ABB RAPID module: Rob2_MainModule.mod

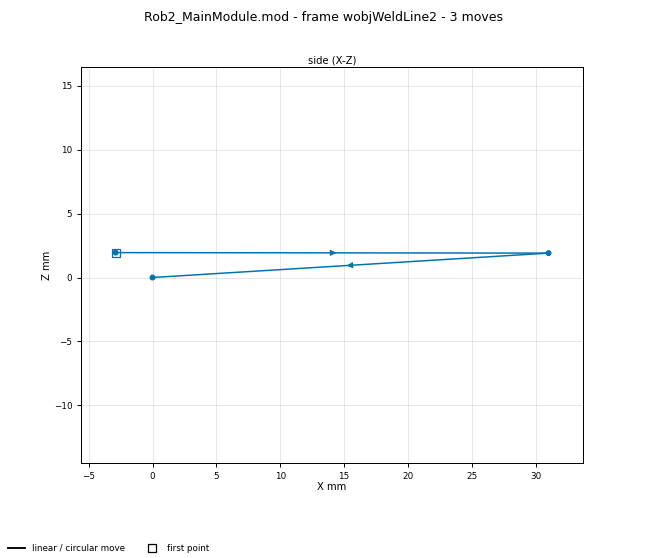
[picture p0: tool path of Rob2_MainModule.mod in frame wobjWeldLine2, 3 of 41 moves have a stored position in this frame; points joined in program order, loops and branches not executed]
MODULE Rob2_MainModule
	!========================================
	! TASK2 (Robot2) - Rob2_MainModule
	! Version History
	!========================================
	! v1.9.44 (2026-02-24) - FIX: Restore MoveAbsJ in MoveJgJ for home return
	!   - ROOT CAUSE: v1.9.42 removed robot motion from MoveJgJ
	!     T_Head rMoveToRobotHome sends robot joint targets via jRob2 PERS
	!     but Robot2 ignored them, causing home return to not move robots
	!   - FIX: MoveAbsJ jRob2, vSync, fine, tool0 restored
	!     MoveAbsJ is joint-space; tool0 vs tWeld2 does not affect joint angles
	!     MergeJgWith() defaults to CJointT for unspecified axes (backward compatible)
	!
	! v1.9.43 (2026-02-21) - Floor coordinate TCP logging
	!   - Added CRobT(\Tool:=tWeld2\WObj:=WobjFloor) to SetRobot2InitialPosition
	!   - Logs TCP_Floor position + orientation to robot2_init_position.txt
	!   - For verifying Robot1/Robot2 TCP meeting point at R-axis center
	!
	! v1.9.42 (2026-02-19) - MoveJgJ fix for tWeld2 [REVERTED in v1.9.44]
	!   - Removed MoveAbsJ jRob2 from MoveJgJ case
	!   - jRob2.robax is tool0-calculated (138deg J2 change from tWeld2 HOME)
	!   - Robot2 now immediately Acks without moving during gantry move
	!   - Prevents concurrent MoveAbsJ conflict with Robot1
	!
	! v2.1.0 (2026-02-03)
	!   - Added PlanA-style command monitoring loop
	!   - Robot2_CommandLoop() monitors nCmdInput from ConfigModule
	!   - TEST_MODE=10 enters real-time command monitoring
	!   - Responds to CMD_WELD, CMD_EDGE_WELD, CMD_ROB2_WIRE_CUT
	!
	! v1.0.0 (2025-12-17)
	!   - Initial gantry position sharing system
	!   - Added shared_gantry_pos and related variables
	!   - Created UpdateSharedGantryPosition procedure
	!
	! v1.1.0 (2025-12-18)
	!   - Added wobj0 definition verification
	!   - Verified Robot2's wobj0 is READ-ONLY (equals World)
	!   - Documented wobj0 vs WobjFloor relationship
	!
	! v1.2.0 (2025-12-18)
	!   - Added WobjFloor coordinate system
	!   - Frame: [-9500, 5300, 2100] with quaternion [0, 1, 0, 0]
	!   - Quaternion [0,1,0,0] = 180deg rotation around X-axis (Y,Z inverted)
	!   - Added comprehensive coordinate system documentation
	!
	! v1.3.0 (2025-12-18)
	!   - Added coordinate verification procedures
	!   - TestRobot2_TCP: TCP position verification in wobj0 and WobjFloor
	!   - TestRobot2_XYZ: X/Y/Z axis movement tests
	!   - TestCoordinateMovement: Core movement and logging procedure
	!   - WritePosToFile: File logging with overwrite mode
	!
	! v1.4.0 (2025-12-18)
	!   - Added World coordinate comparison
	!   - CompareRobot2Coordinates: Compare wobj0, WobjFloor, World
	!   - Verified relationship: wobj0 = World (for Robot2)
	!   - Verified WobjFloor transforms coordinates correctly
	!
	! v1.4.1 (2025-12-23)
	!   - Removed MoveToMiddlePosition calls to prevent Reference Error
	!   - Simplified procedure calls in TestRobot2_TCP
	!
	! v1.4.2 (2025-12-24)
	!   - Added Robot2 TCP coordinate movement tests
	!   - TestCoordinateMovement: Move and log TCP positions
	!
	! v1.4.3 (2025-12-24)
	!   - Combined X/Y/Z tests into single TestRobot2_XYZ procedure
	!   - Streamlined coordinate testing workflow
	!
	! v1.4.4 (2025-12-24)
	!   - Reduced movement distance to avoid joint limits
	!   - Changed test distances: 50mm X, 30mm Y, 20mm Z
	!
	! v1.4.5 (2025-12-24)
	!   - Increased movement back to 50/30/20 mm
	!   - Added return to start position after test
	!
	! v1.4.6 (2025-12-24)
	!   - Added home position test capability
	!   - Save original joint position with CJointT()
	!   - Move to home position [0,0,0,0,0,0] before test
	!   - Return to original position after test
	!
	! v1.4.7 (2025-12-24)
	!   - Fixed singularity error in home position
	!   - Changed Robot2 home position to [+90,0,0,0,30,0]
	!   - J1=+90deg for Robot2 mounting orientation
	!   - J5=30deg to avoid wrist singularity (not 0deg)
	!
	! v1.5.0 (2025-12-24) - DUAL COORDINATE SYSTEM
	!   - Added config.txt MODE support for dual coordinate systems
	!   - ReadConfigMode() function reads /HOME/config.txt
	!   - MODE=0 (Default - User's system):
	!     * Robot2 uses WobjFloor as base coordinate
	!     * wobj0 [+50,+30,+20] -> Floor [+50,+30,+20] (NO Y,Z inversion)
	!   - MODE=1 (Claude's system):
	!     * Robot2 uses wobj0 as base coordinate
	!     * wobj0 [+50,+30,+20] -> Floor [+50,-30,-20] (Y,Z inverted)
	!   - Modified TestCoordinateMovement to accept wobjdata parameter
	!   - TestRobot2_XYZ now switches coordinate system based on MODE
	!
	! v1.7.45 - v1.7.47 (2025-12-31)
	!   - Updated SetRobot2InitialPosition to match Robot1 HOME position
	!   - Robot2 HOME: TCP [0, 488, -1000] with quaternion [0.50000, -0.50000, -0.50000, -0.50000]
	!   - Fixed 40512 error using actual extax values from CJointT()
	!
	! v1.7.50 (2025-12-31)
	!   - Added WobjGantry_Rob2 dynamic work object for Robot2 TCP control
	!   - Implemented UpdateGantryWobj_Rob2() to read gantry position from TASK1
	!   - Robot2 cannot control gantry - must use CJointT(\TaskName:="T_ROB1")
	!   - R-axis rotation with 90deg base offset (R=0: gantry parallel to Y-axis)
	!   - Enables Robot2 TCP control in Floor coordinates regardless of gantry position
	!   - SetRobot2InitialPosition now uses WobjGantry_Rob2 instead of wobj0
	!========================================

    RECORD targetdata
        robtarget position;
        num cpm;
        num schedule;
        num voltage;
        num wfs;
        num Current;
        num WeaveShape;
        num WeaveType;
        num WeaveLength;
        num WeaveWidth;
        num WeaveDwellLeft;
        num WeaveDwellRight;
        num TrackType;
        num TrackGainY;
        num TrackGainZ;
        num MaxCorr;
        num Bias;
    ENDRECORD

    RECORD monRobs
        extjoint monExt;
        robjoint monJoint1;
        robjoint monJoint2;
        pose monPose1;
        pose monPose2;
    ENDRECORD

    RECORD torchmotion
        num No;
        num LengthOffset;
        num BreadthOffset;
        num HeightOffset;
        num WorkingAngle;
        num TravelAngle;
        num WeldingSpeed;
        num Schedule;
        num Voltage;
        num FeedingSpeed;
        num Current;
        num WeaveShape;
        num WeaveType;
        num WeaveLength;
        num WeaveWidth;
        num WeaveDwellLeft;
        num WeaveDwellRight;
        num TrackType;
        num TrackGainY;
        num TrackGainZ;
        num MaxCorr;
        num Bias;
    ENDRECORD

    RECORD corrorder
        num X_StartOffset;
        num X_Depth;
        num X_ReturnLength;
        num Y_StartOffset;
        num Y_Depth;
        num Y_ReturnLength;
        num Z_StartOffset;
        num Z_Depth;
        num Z_ReturnLength;
        num RY_Torch;
    ENDRECORD

    RECORD edgedata
        pos EdgePos;
        num Height;
        num Breadth;
        num HoleSize;
        num Thickness;
        num AngleHeight;
        num AngleWidth;
    ENDRECORD

	! v1.7.51 (2026-01-03)
	!   - Added robot2_init_complete synchronization flag
	!   - TASK2 sets flag to TRUE after SetRobot2InitialPosition completes
	!   - Enables precise TASK1/TASK2 synchronization without fixed delays
	!   - Replaces crude WaitTime 10.0 approach with event-based signaling
	!
	! v1.8.0 (2026-01-03)
	!   - Version sync with TASK1 for R-axis rotation testing
	!   - No functional changes in TASK2 (changes in TASK1 only)
	!   - Ready for Phase 2: Complex motion testing
	!
	! v1.8.7 (2026-01-05)
	!   - FIX: Use gantry extax from TASK1 for Robot2 MoveJ/MoveL in SetRobot2InitialPosition.
	!
	! v1.8.9 (2026-01-05)
	!   - STABILITY: Reduced TPWrite output and file writes in SetRobot2InitialPosition.
	!
	! v1.8.10 (2026-01-05)
	!   - FEAT: Added TEST_MODE=2 Robot2 TCP offset move from config.txt.
	!
	! v1.8.11 (2026-01-06)
	!   - FIX: Guard config parsing in SetRobot2OffsetPosition to avoid StrPart errors.
	!
	! v1.8.12 (2026-01-06)
	!   - FIX: Allow missing TCP_OFFSET_* with default 0 values.
	!
	! v1.8.13 (2026-01-06)
	!   - Version sync with TASK1 (Mode2 range checks).
	!
	! v1.8.14 (2026-01-06)
	!   - Version sync with TASK1 (MOC.cfg range update).
	!
	! v1.8.15 (2026-01-06)
	!   - FIX: Use TASK PERS for robot1_floor_pos_t2 to avoid global PERS ambiguity.
	!
	! v1.8.16 (2026-01-06)
	!   - FIX: Initialize TASK PERS robot1_floor_pos_t2 to satisfy RAPID syntax.
	!
	! v1.8.18 (2026-01-06)
	!   - Version sync with TASK1 (robot1_floor_pos_t1 rename in TASK1).
	!
	! v1.8.19 (2026-01-06)
	!   - Version sync with TASK1 (robot2_floor_pos_t1 rename in TASK1).
	!
	! v1.8.20 (2026-01-06)
	!   - FIX: Rename robot2_floor_pos to robot2_floor_pos_t1 and remove initializer.
	!
	! v1.8.21 (2026-01-06)
	!   - Version sync with TASK1 (Mode2 gantry HOME return).
	!
	! v1.8.22 (2026-01-06)
	!   - FEAT: Support per-robot TCP offsets (R2) for Mode2 via TCP_OFFSET_R2_*.
	!
	! v1.8.23 (2026-01-07)
	!   - FIX: Make Mode2 TCP offset parsing tolerant of leading whitespace.
	!
	! v1.8.24 (2026-01-07)
	!   - Version sync with TASK1 (Mode2 TCP offset debug logging).
	!
	! v1.8.25 (2026-01-07)
	!   - Version sync with TASK1 (ignore comment lines during offset parse).
	!
	! v1.8.26 (2026-01-07)
	!   - Version sync with TASK1 (trim leading whitespace during offset parse).
	!
	! v1.8.27 (2026-01-07)
	!   - Version sync with TASK1 (remove tab escape in trim loop).
	!
	! v1.8.28 (2026-01-07)
	!   - Version sync with TASK1 (remove RemoveCR in offset parse loop).
	!
	! v1.8.29 (2026-01-07)
	!   - Version sync with TASK1 (remove RemoveCR in offset parse loop).
	!
! v1.8.31 (2026-01-07)
!   - FIX: Use TASK PERS for robot2_init_complete to share flag with TASK1.
!   - FIX: Set robot2_init_complete right after Step1 to avoid TASK1 timeout.
!   - FIX: Add EOF-safe config parsing in ReadTestMode and Mode2 offset parse.
!   - DIAG: Log Mode2 offset start in main process.
!
! v1.8.32 (2026-01-08)
!   - Version sync with TASK1 (robot2_init_complete init in TASK1).
!
! v1.8.33 (2026-01-08)
!   - DIAG: Log entry at start of TASK2 main before config read.
!
! v1.8.34 (2026-01-08)
!   - DIAG: Bypass ReadTestMode temporarily (force TEST_MODE=2).
!
! v1.8.35 (2026-01-08)
!   - FIX: Revert robot2_init_complete to shared PERS for cross-task sync.
!
! v1.8.36 (2026-01-08)
!   - DIAG: Log Mode2 offset inputs, gantry extax, and target TCP before MoveJ.
!
! v1.8.37 (2026-01-08)
!   - DIAG: Create Mode2 offset log at entry before config parsing.
!
! v1.8.38 (2026-01-08)
!   - FIX: Guard comment detection to avoid StrPart on empty strings in config parse.
!
! v1.8.39 (2026-01-08)
!   - FIX - Read Mode2 TCP offsets from TASK1 shared PERS (no config read).
!
! v1.8.55 (2026-01-12)
!   - FIX - Remove 488mm from offset_tcp calculation
!   - CAUSE - MoveJ uses WobjGantry_Rob2 (R-center reference)
!   - 488mm was only needed for wobj0 reference, not WobjGantry_Rob2
!   - RESULT - TCP distance 200mm fixed (R-angle independent)
	!
	! v1.8.30 (2026-01-07)
	!   - Version sync with TASK1 (stop offset parse once keys are found).
	!
	! v1.8.17 (2026-01-06)
	!   - FIX: Rename TASK2 local copy to robot1_floor_pos_t2 to avoid PERS ambiguity.
	!
	! v1.8.8 (2026-01-05)
	!   - STABILITY: Reduced main process log writes to lower 41617 risk.
	!
	! v1.8.5 (2026-01-04)
	!   - Version synchronized with TASK1 (Robot2 angle correction in TASK1).
	!   - No functional changes in TASK2.
	!
	! v1.8.3 (2026-01-04)
	!   - STABILITY: Added ERROR handlers to main and SetRobot2InitialPosition
	!   - STABILITY: Corrected file handle usage in 4 procedures (single Open statement)
	!   - STANDARDS: Replaced Unicode characters (deg symbol) with ASCII equivalents
	!   - STANDARDS: Changed file encoding from UTF-8 to ASCII
	!   - Version synchronized with TASK1 (jumped from v1.8.0)
	!
! Version constant for logging (v1.8.39+)
CONST string TASK2_VERSION := "v1.9.46";

! Synchronization flag for TASK1/TASK2 initialization
! TASK2 sets this to TRUE when Robot2 initialization is complete
! TASK1 waits for this flag before starting gantry floor tests
PERS bool robot2_init_complete;
! Mode2 TCP offsets for Robot2 (shared from TASK1)
PERS num mode2_r2_offset_x;
PERS num mode2_r2_offset_y;
PERS num mode2_r2_offset_z;

! v1.8.57: Synchronization flag - wait for TASK1 to update config values
PERS bool mode2_config_ready;

! v1.8.63: Robot2 reposition sync flags
PERS bool mode2_r2_reposition_trigger;
PERS bool mode2_r2_reposition_done;
! v1.8.67: Initial offset complete flag
PERS bool mode2_r2_initial_offset_done;

! v1.9.17: Shared test_mode from TASK1
PERS num shared_test_mode;

! v2.1.0: Command Interface Variables (shared with TASK1 ConfigModule)
PERS num nCmdInput;
PERS num nCmdOutput;
PERS num nCmdMatch;

! v2.1.0: Command Constants (must match TASK1 ConfigModule)
CONST num CMD_MOVE_TO_WORLDHOME := 101;
CONST num CMD_WELD := 200;
CONST num CMD_WELD_MOTION := 201;
CONST num CMD_EDGE_WELD := 210;
CONST num CMD_ROB2_WIRE_CUT := 512;

! v1.8.70: Store Robot2 offset joints (like robot1_offset_joints in TASK1)
! Initial call: MoveJ then save joints
! Reposition call: Skip MoveJ (joints already at offset, gantry moved)
VAR robjoint robot2_offset_joints;

    PERS tasks taskGroup12{2};
    PERS tasks taskGroup13{2};
    PERS tasks taskGroup23{2};
    PERS tasks taskGroup123{3};
    PERS pos nCaledR2Pos;
    TASK PERS jointtarget jTemp:=[[0,-2.51761,-12.1411,0,15.6587,0],[-500,500,300,15,0,-28.6479]];
    PERS wobjdata wobjtest:=[FALSE,TRUE,"GantryRob",[[-971.372,373.696,300],[1,0,0,0]],[[0,0,0],[1,0,0,0]]];

    ! Sync Data
    TASK VAR syncident SynchronizeJGJon{9999};
    TASK VAR syncident SynchronizePGJon{9999};
    TASK VAR syncident SynchronizePGLon{9999};
    TASK VAR syncident SynchronizeJGJoff{9999};
    TASK VAR syncident SynchronizePGJoff{9999};
    TASK VAR syncident SynchronizePGLoff{9999};
    TASK VAR syncident Wait{100};

    PERS string stCommand;
    PERS string stReact{3};
    PERS num idSync;
    PERS speeddata vSync;
    PERS zonedata zSync;

    PERS wobjdata wobjWeldLine2;
    PERS wobjdata wobjRotCtr2;

    ! Weld Sequence Sync Variables (v1.9.0)
    ! Cross-task synchronization with TASK1
    PERS bool t2_weld_ready;    ! Robot2 ready signal (set by TASK2)
    PERS bool t1_weld_start;    ! TASK1 weld start signal (read by TASK2)
    PERS bool t1_weld_done;     ! TASK1 weld done signal (read by TASK2)

    ! Edge-based Weld Sequence Sync Variables (v2.0.0)
    ! From TASK1 MainModule
    PERS bool t1_weld_position_ready;  ! TASK1 gantry+Robot1 positioned
    PERS bool shared_bRobSwap;         ! Robot swap flag from TASK1

    ! Robot2 edge positions (shared from TASK1, v1.9.37)
    PERS pos shared_posStart_r2;
    PERS pos shared_posEnd_r2;
    PERS num shared_nLengthWeldLine;

    ! stCommand/stReact Protocol (v1.9.39 - T_Head interface)
    ! T_Head sets stCommand, TASK1/2 respond via stReact
    ! NOTE: stCommand/stReact already declared above (lines 361-362)

    ! Weld WObj for Robot2 (v1.9.0)
    ! Created by TASK1, referenced by TASK2
    PERS wobjdata WobjWeldR2;

    ! Robot2 Weld Orientation from ConfigModule (v1.9.0)
    ! Cross-task reference to TASK1 ConfigModule
    PERS num WELD_R2_ORIENT_Q1;
    PERS num WELD_R2_ORIENT_Q2;
    PERS num WELD_R2_ORIENT_Q3;
    PERS num WELD_R2_ORIENT_Q4;

    ! Robot2 Weld Position in WObj (v1.9.1)
    ! Cross-task reference to TASK1 ConfigModule
    ! WObj: X=weld direction, Y=perpendicular, Z=Floor Z
    PERS num WELD_R2_WObj_X;
    PERS num WELD_R2_WObj_Y;
    PERS num WELD_R2_WObj_Z;

    ! Work Object Definitions (v1.7.13 2025-12-28)
    ! WobjFloor: Floor coordinate system from TASK1 (external reference)
    PERS wobjdata WobjFloor;

    ! WobjFloor_Rob2: Floor coordinate system for Robot2
    ! MUST be identical to TASK1's WobjFloor (absolute world coordinate)
    ! uframe: [-9500, 5300, 2100] = Gantry HOME in Floor coordinate
    ! rot: [1, 0, 0, 0] = No rotation (Robot2 wobj0 aligned with Floor!)
    PERS wobjdata WobjFloor_Rob2 := [FALSE, TRUE, "", [[-9500, 5300, 2100], [1, 0, 0, 0]], [[0, 0, 0], [1, 0, 0, 0]]];

    ! WobjGantry_Rob2: Dynamic work object for Robot2 TCP control (v1.7.50)
    ! Updated by UpdateGantryWobj_Rob2() to track gantry position from TASK1
    ! Allows Robot2 TCP control in Floor coordinates regardless of gantry position
    ! Robot2 cannot control gantry, must read position from TASK1
    PERS wobjdata WobjGantry_Rob2 := [FALSE, TRUE, "", [[0, 0, 0], [1, 0, 0, 0]], [[0, 0, 0], [1, 0, 0, 0]]];

    ! WobjRobot2Base_Dynamic: Robot2 base coordinate from TASK1 (external reference) (v1.7.50)
    ! TASK1 updates this to track Robot2 base position as gantry moves
    ! Robot2 uses this to calculate its Floor TCP position
    ! Direction = Floor direction (no rotation, quaternion [1,0,0,0])
    PERS wobjdata WobjRobot2Base_Dynamic;

    ! wobjRob2Base: Robot2 Base Frame orientation from MOC.cfg
    ! Quaternion [-4.32964E-17, 0.707107, 0.707107, 4.32964E-17] = 45deg rotation
    PERS wobjdata wobjRob2Base := [FALSE, TRUE, "", [[0, 0, 0], [-0.0000000000000000432964, 0.707107, 0.707107, 0.0000000000000000432964]], [[0, 0, 0], [1, 0, 0, 0]]];

    ! Robot Position Monitoring (v1.5.1 2025-12-25)
    ! Robot1 TCP position from TASK1 (local copy for TASK2)
    TASK PERS robtarget robot1_floor_pos_t2 := [[0,0,0],[1,0,0,0],[0,0,0,0],[0,0,0,0,0,0]];
    ! Robot1 wobj0 snapshot from TASK1 (external reference)
    PERS wobjdata robot1_wobj0_snapshot := [FALSE, TRUE, "", [[0,0,0],[1,0,0,0]], [[0,0,0],[1,0,0,0]]];

    ! Robot2 TCP position in Floor coordinate system (for distance measurement)
    ! Shared across tasks - use PERS (not TASK PERS) for cross-task access
    PERS robtarget robot2_floor_pos_t1;

    PERS num nMotionTotalStep{2};
    PERS num nMotionStepCount{2};
    PERS num nMotionStartStepLast{2};
    PERS num nMotionEndStepLast{2};
    PERS num nRunningStep{2};
    PERS num nWeldSequence;

    PERS jointtarget jRob2;
    PERS robtarget pRob2;
    PERS bool bRqMoveG_PosHold;

    PERS robtarget pctWeldPosR1;
    PERS robtarget pctWeldPosR2;

    PERS targetdata Welds2{40};
    TASK PERS speeddata vWeld{40}:=[[10,200,200,200],[10,200,200,200],[10,200,200,200],[10,200,200,200],[9.16667,200,200,200],[9.16667,200,200,200],[8.33333,200,200,200],[7.5,200,200,200],[0,0,0,0],[0,0,0,0],[0,0,0,0],[0,0,0,0],[0,0,0,0],[0,0,0,0],[0,0,0,0],[0,0,0,0],[0,0,0,0],[0,0,0,0],[0,0,0,0],[0,0,0,0],[0,0,0,0],[0,0,0,0],[0,0,0,0],[0,0,0,0],[0,0,0,0],[0,0,0,0],[0,0,0,0],[0,0,0,0],[0,0,0,0],[0,0,0,0],[0,0,0,0],[0,0,0,0],[0,0,0,0],[0,0,0,0],[0,0,0,0],[0,0,0,0],[0,0,0,0],[0,0,0,0],[0,0,0,0],[10,200,200,200]];
    PERS seamdata smDefault_2{2};


    PERS speeddata vTargetSpeed;
    PERS zonedata zTargetZone;

    TASK PERS welddata wdTrap:=[10,0,[5,0,38,240,0,400,0,0,0],[0,0,0,0,0,0,0,0,0]];
    TASK PERS welddata wd1:=[10,0,[5,0,39.5,260,0,0,0,0,0],[0,0,0,0,0,0,0,0,0]];
    TASK PERS welddata wd2:=[10,0,[5,0,39.5,260,0,0,0,0,0],[0,0,0,0,0,0,0,0,0]];
    TASK PERS welddata wd3:=[10,0,[5,0,39.5,260,0,0,0,0,0],[0,0,0,0,0,0,0,0,0]];
    TASK PERS welddata wd4:=[10,0,[5,0,39.5,260,0,0,0,0,0],[0,0,0,0,0,0,0,0,0]];
    TASK PERS welddata wd5:=[9.16667,0,[5,0,39.5,255,0,420,0,0,0],[0,0,0,0,0,0,0,0,0]];
    TASK PERS welddata wd6:=[9.16667,0,[5,0,39.5,255,0,420,0,0,0],[0,0,0,0,0,0,0,0,0]];
    TASK PERS welddata wd7:=[8.33333,0,[5,0,39.5,255,0,420,0,0,0],[0,0,0,0,0,0,0,0,0]];
    TASK PERS welddata wd8:=[7.5,0,[5,0,36,225,0,375,0,0,0],[0,0,0,0,0,0,0,0,0]];
    TASK PERS welddata wd9:=[7.5,0,[5,0,36,225,0,375,0,0,0],[0,0,0,0,0,0,0,0,0]];
    TASK PERS welddata wd10:=[0,0,[5,0,0,0,0,0,0,0,0],[0,0,0,0,0,0,0,0,0]];
    TASK PERS welddata wd11:=[0,0,[5,0,0,0,0,0,0,0,0],[0,0,0,0,0,0,0,0,0]];
    TASK PERS welddata wd12:=[0,0,[5,0,0,0,0,0,0,0,0],[0,0,0,0,0,0,0,0,0]];
    TASK PERS welddata wd13:=[0,0,[5,0,0,0,0,0,0,0,0],[0,0,0,0,0,0,0,0,0]];
    TASK PERS welddata wd14:=[0,0,[5,0,0,0,0,0,0,0,0],[0,0,0,0,0,0,0,0,0]];
    TASK PERS welddata wd15:=[0,0,[5,0,0,0,0,0,0,0,0],[0,0,0,0,0,0,0,0,0]];
    TASK PERS welddata wd16:=[0,0,[5,0,0,0,0,0,0,0,0],[0,0,0,0,0,0,0,0,0]];
    TASK PERS welddata wd17:=[0,0,[5,0,0,0,0,0,0,0,0],[0,0,0,0,0,0,0,0,0]];
    TASK PERS welddata wd18:=[0,0,[5,0,0,0,0,0,0,0,0],[0,0,0,0,0,0,0,0,0]];
    TASK PERS welddata wd19:=[0,0,[5,0,0,0,0,0,0,0,0],[0,0,0,0,0,0,0,0,0]];
    TASK PERS welddata wd20:=[0,0,[5,0,0,0,0,0,0,0,0],[0,0,0,0,0,0,0,0,0]];
    TASK PERS welddata wd21:=[0,0,[5,0,0,0,0,0,0,0,0],[0,0,0,0,0,0,0,0,0]];
    TASK PERS welddata wd22:=[0,0,[5,0,0,0,0,0,0,0,0],[0,0,0,0,0,0,0,0,0]];
    TASK PERS welddata wd23:=[0,0,[5,0,0,0,0,0,0,0,0],[0,0,0,0,0,0,0,0,0]];
    TASK PERS welddata wd24:=[0,0,[5,0,0,0,0,0,0,0,0],[0,0,0,0,0,0,0,0,0]];
    TASK PERS welddata wd25:=[0,0,[5,0,0,0,0,0,0,0,0],[0,0,0,0,0,0,0,0,0]];
    TASK PERS welddata wd26:=[0,0,[5,0,0,0,0,0,0,0,0],[0,0,0,0,0,0,0,0,0]];
    TASK PERS welddata wd27:=[0,0,[5,0,0,0,0,0,0,0,0],[0,0,0,0,0,0,0,0,0]];
    TASK PERS welddata wd28:=[0,0,[5,0,0,0,0,0,0,0,0],[0,0,0,0,0,0,0,0,0]];
    TASK PERS welddata wd29:=[0,0,[5,0,0,0,0,0,0,0,0],[0,0,0,0,0,0,0,0,0]];
    TASK PERS welddata wd30:=[0,0,[5,0,0,0,0,0,0,0,0],[0,0,0,0,0,0,0,0,0]];
    TASK PERS welddata wd31:=[0,0,[5,0,0,0,0,0,0,0,0],[0,0,0,0,0,0,0,0,0]];
    TASK PERS welddata wd32:=[0,0,[5,0,0,0,0,0,0,0,0],[0,0,0,0,0,0,0,0,0]];
    TASK PERS welddata wd33:=[0,0,[5,0,0,0,0,0,0,0,0],[0,0,0,0,0,0,0,0,0]];
    TASK PERS welddata wd34:=[0,0,[5,0,0,0,0,0,0,0,0],[0,0,0,0,0,0,0,0,0]];
    TASK PERS welddata wd35:=[0,0,[5,0,0,0,0,0,0,0,0],[0,0,0,0,0,0,0,0,0]];
    TASK PERS welddata wd36:=[0,0,[5,0,0,0,0,0,0,0,0],[0,0,0,0,0,0,0,0,0]];
    TASK PERS welddata wd37:=[0,0,[5,0,0,0,0,0,0,0,0],[0,0,0,0,0,0,0,0,0]];
    TASK PERS welddata wd38:=[0,0,[5,0,0,0,0,0,0,0,0],[0,0,0,0,0,0,0,0,0]];
    TASK PERS welddata wd39:=[0,0,[5,0,0,0,0,0,0,0,0],[0,0,0,0,0,0,0,0,0]];
    TASK PERS welddata wd40:=[10,0,[5,0,39.5,260,0,0,0,0,0],[0,0,0,0,0,0,0,0,0]];

    TASK PERS welddata Holdwd1:=[0.01,0,[5,0,39.5,260,0,0,0,0,0],[0,0,0,0,0,0,0,0,0]];
    TASK PERS welddata Holdwd2:=[0.01,0,[5,0,39.5,260,0,0,0,0,0],[0,0,0,0,0,0,0,0,0]];
    TASK PERS welddata Holdwd3:=[0.01,0,[5,0,39.5,260,0,0,0,0,0],[0,0,0,0,0,0,0,0,0]];
    TASK PERS welddata Holdwd4:=[0.01,0,[5,0,39.5,260,0,0,0,0,0],[0,0,0,0,0,0,0,0,0]];
    TASK PERS welddata Holdwd5:=[0.01,0,[5,0,39.5,255,0,420,0,0,0],[0,0,0,0,0,0,0,0,0]];
    TASK PERS welddata Holdwd6:=[0.01,0,[5,0,39.5,255,0,420,0,0,0],[0,0,0,0,0,0,0,0,0]];
    TASK PERS welddata Holdwd7:=[0.01,0,[5,0,39.5,255,0,420,0,0,0],[0,0,0,0,0,0,0,0,0]];
    TASK PERS welddata Holdwd8:=[0.01,0,[5,0,36,225,0,375,0,0,0],[0,0,0,0,0,0,0,0,0]];
    TASK PERS welddata Holdwd9:=[0.01,0,[5,0,36,225,0,375,0,0,0],[0,0,0,0,0,0,0,0,0]];
    TASK PERS welddata Holdwd10:=[0.01,0,[5,0,0,0,0,0,0,0,0],[0,0,0,0,0,0,0,0,0]];

    !!! weave data !!!
    TASK PERS weavedata weaveTrap:=[1,2,3,3,0,0,0,0,0,0,0,0,0,0,0];
    TASK PERS weavedata weave1:=[1,2,2,3,0,0,0,0,0,0,0,0,0,0,0];
    TASK PERS weavedata weave2:=[1,2,2,3,0,0,0,0,0,0,0,0,0,0,0];
    TASK PERS weavedata weave3:=[1,2,2,3,0,0,0,0,0,0,0,0,0,0,0];
    TASK PERS weavedata weave4:=[1,2,2,3,0,0,0,0,0,0,0,0,0,0,0];
    TASK PERS weavedata weave5:=[1,2,2,3.5,0,0,0,0,0,0,0,0,0,0,0];
    TASK PERS weavedata weave6:=[1,2,2,3.5,0,0,0,0,0,0,0,0,0,0,0];
    TASK PERS weavedata weave7:=[1,2,2,3.5,0,0,0,0,0,0,0,0,0,0,0];
    TASK PERS weavedata weave8:=[1,0,0,0,0,0,0,0,0,0,0,0,0,0,0];
    TASK PERS weavedata weave9:=[1,0,0,0,0,0,0,0,0,0,0,0,0,0,0];
    TASK PERS weavedata weave10:=[0,0,0,0,0,0,0,0,0,0,0,0,0,0,0];
    TASK PERS weavedata weave11:=[0,0,0,0,0,0,0,0,0,0,0,0,0,0,0];
    TASK PERS weavedata weave12:=[0,0,0,0,0,0,0,0,0,0,0,0,0,0,0];
    TASK PERS weavedata weave13:=[0,0,0,0,0,0,0,0,0,0,0,0,0,0,0];
    TASK PERS weavedata weave14:=[0,0,0,0,0,0,0,0,0,0,0,0,0,0,0];
    TASK PERS weavedata weave15:=[0,0,0,0,0,0,0,0,0,0,0,0,0,0,0];
    TASK PERS weavedata weave16:=[0,0,0,0,0,0,0,0,0,0,0,0,0,0,0];
    TASK PERS weavedata weave17:=[0,0,0,0,0,0,0,0,0,0,0,0,0,0,0];
    TASK PERS weavedata weave18:=[0,0,0,0,0,0,0,0,0,0,0,0,0,0,0];
    TASK PERS weavedata weave19:=[0,0,0,0,0,0,0,0,0,0,0,0,0,0,0];
    TASK PERS weavedata weave20:=[0,0,0,0,0,0,0,0,0,0,0,0,0,0,0];
    TASK PERS weavedata weave21:=[0,0,0,0,0,0,0,0,0,0,0,0,0,0,0];
    TASK PERS weavedata weave22:=[0,0,0,0,0,0,0,0,0,0,0,0,0,0,0];
    TASK PERS weavedata weave23:=[0,0,0,0,0,0,0,0,0,0,0,0,0,0,0];
    TASK PERS weavedata weave24:=[0,0,0,0,0,0,0,0,0,0,0,0,0,0,0];
    TASK PERS weavedata weave25:=[0,0,0,0,0,0,0,0,0,0,0,0,0,0,0];
    TASK PERS weavedata weave26:=[0,0,0,0,0,0,0,0,0,0,0,0,0,0,0];
    TASK PERS weavedata weave27:=[0,0,0,0,0,0,0,0,0,0,0,0,0,0,0];
    TASK PERS weavedata weave28:=[0,0,0,0,0,0,0,0,0,0,0,0,0,0,0];
    TASK PERS weavedata weave29:=[0,0,0,0,0,0,0,0,0,0,0,0,0,0,0];
    TASK PERS weavedata weave30:=[0,0,0,0,0,0,0,0,0,0,0,0,0,0,0];
    TASK PERS weavedata weave31:=[0,0,0,0,0,0,0,0,0,0,0,0,0,0,0];
    TASK PERS weavedata weave32:=[0,0,0,0,0,0,0,0,0,0,0,0,0,0,0];
    TASK PERS weavedata weave33:=[0,0,0,0,0,0,0,0,0,0,0,0,0,0,0];
    TASK PERS weavedata weave34:=[0,0,0,0,0,0,0,0,0,0,0,0,0,0,0];
    TASK PERS weavedata weave35:=[0,0,0,0,0,0,0,0,0,0,0,0,0,0,0];
    TASK PERS weavedata weave36:=[0,0,0,0,0,0,0,0,0,0,0,0,0,0,0];
    TASK PERS weavedata weave37:=[0,0,0,0,0,0,0,0,0,0,0,0,0,0,0];
    TASK PERS weavedata weave38:=[0,0,0,0,0,0,0,0,0,0,0,0,0,0,0];
    TASK PERS weavedata weave39:=[0,0,0,0,0,0,0,0,0,0,0,0,0,0,0];
    TASK PERS weavedata weave40:=[1,2,2,3,0,0,0,0,0,0,0,0,0,0,0];

    !!! Track Data !!!
    TASK PERS trackdata trackTrap:=[0,FALSE,50,[0,0,0,0,0,0,0,0,0],[0,0,0,0,0,0,0]];
    TASK PERS trackdata track0:=[0,FALSE,50,[0,0,0,0,0,0,0,0,0],[0,0,0,0,0,0,0]];
    TASK PERS trackdata track1:=[0,FALSE,50,[0,0,0,0,0,0,0,0,0],[0,0,0,0,0,0,0]];
    TASK PERS trackdata track2:=[0,FALSE,50,[0,0,0,0,0,0,0,0,0],[0,0,0,0,0,0,0]];
    TASK PERS trackdata track3:=[0,FALSE,50,[0,0,0,0,0,0,0,0,0],[0,0,0,0,0,0,0]];
    TASK PERS trackdata track4:=[0,FALSE,50,[0,0,0,0,0,0,0,0,0],[0,0,0,0,0,0,0]];
    TASK PERS trackdata track5:=[0,FALSE,50,[0,0,0,0,0,0,0,0,0],[0,0,0,0,0,0,0]];
    TASK PERS trackdata track6:=[0,FALSE,50,[0,0,0,0,0,0,0,0,0],[0,0,0,0,0,0,0]];
    TASK PERS trackdata track7:=[0,FALSE,50,[0,0,0,0,0,0,0,0,0],[0,0,0,0,0,0,0]];
    TASK PERS trackdata track8:=[0,FALSE,50,[0,0,0,0,0,0,0,0,0],[0,0,0,0,0,0,0]];
    TASK PERS trackdata track9:=[0,FALSE,50,[0,0,0,0,0,0,0,0,0],[0,0,0,0,0,0,0]];
    TASK PERS trackdata track10:=[0,FALSE,50,[0,0,0,0,0,0,0,0,0],[0,0,0,0,0,0,0]];
    TASK PERS trackdata track11:=[0,FALSE,50,[0,0,0,0,0,0,0,0,0],[0,0,0,0,0,0,0]];
    TASK PERS trackdata track12:=[0,FALSE,50,[0,0,0,0,0,0,0,0,0],[0,0,0,0,0,0,0]];
    TASK PERS trackdata track13:=[0,FALSE,50,[0,0,0,0,0,0,0,0,0],[0,0,0,0,0,0,0]];
    TASK PERS trackdata track14:=[0,FALSE,50,[0,0,0,0,0,0,0,0,0],[0,0,0,0,0,0,0]];
    TASK PERS trackdata track15:=[0,FALSE,50,[0,0,0,0,0,0,0,0,0],[0,0,0,0,0,0,0]];
    TASK PERS trackdata track16:=[0,FALSE,50,[0,0,0,0,0,0,0,0,0],[0,0,0,0,0,0,0]];
    TASK PERS trackdata track17:=[0,FALSE,50,[0,0,0,0,0,0,0,0,0],[0,0,0,0,0,0,0]];
    TASK PERS trackdata track18:=[0,FALSE,50,[0,0,0,0,0,0,0,0,0],[0,0,0,0,0,0,0]];
    TASK PERS trackdata track19:=[0,FALSE,50,[0,0,0,0,0,0,0,0,0],[0,0,0,0,0,0,0]];
    TASK PERS trackdata track20:=[0,FALSE,50,[0,0,0,0,0,0,0,0,0],[0,0,0,0,0,0,0]];
    TASK PERS trackdata track21:=[0,FALSE,50,[0,0,0,0,0,0,0,0,0],[0,0,0,0,0,0,0]];
    TASK PERS trackdata track22:=[0,FALSE,50,[0,0,0,0,0,0,0,0,0],[0,0,0,0,0,0,0]];
    TASK PERS trackdata track23:=[0,FALSE,50,[0,0,0,0,0,0,0,0,0],[0,0,0,0,0,0,0]];
    TASK PERS trackdata track24:=[0,FALSE,50,[0,0,0,0,0,0,0,0,0],[0,0,0,0,0,0,0]];
    TASK PERS trackdata track25:=[0,FALSE,50,[0,0,0,0,0,0,0,0,0],[0,0,0,0,0,0,0]];
    TASK PERS trackdata track26:=[0,FALSE,50,[0,0,0,0,0,0,0,0,0],[0,0,0,0,0,0,0]];
    TASK PERS trackdata track27:=[0,FALSE,50,[0,0,0,0,0,0,0,0,0],[0,0,0,0,0,0,0]];
    TASK PERS trackdata track28:=[0,FALSE,50,[0,0,0,0,0,0,0,0,0],[0,0,0,0,0,0,0]];
    TASK PERS trackdata track29:=[0,FALSE,50,[0,0,0,0,0,0,0,0,0],[0,0,0,0,0,0,0]];
    TASK PERS trackdata track30:=[0,FALSE,50,[0,0,0,0,0,0,0,0,0],[0,0,0,0,0,0,0]];
    TASK PERS trackdata track31:=[0,FALSE,50,[0,0,0,0,0,0,0,0,0],[0,0,0,0,0,0,0]];
    TASK PERS trackdata track32:=[0,FALSE,50,[0,0,0,0,0,0,0,0,0],[0,0,0,0,0,0,0]];
    TASK PERS trackdata track33:=[0,FALSE,50,[0,0,0,0,0,0,0,0,0],[0,0,0,0,0,0,0]];
    TASK PERS trackdata track34:=[0,FALSE,50,[0,0,0,0,0,0,0,0,0],[0,0,0,0,0,0,0]];
    TASK PERS trackdata track35:=[0,FALSE,50,[0,0,0,0,0,0,0,0,0],[0,0,0,0,0,0,0]];
    TASK PERS trackdata track36:=[0,FALSE,50,[0,0,0,0,0,0,0,0,0],[0,0,0,0,0,0,0]];
    TASK PERS trackdata track37:=[0,FALSE,50,[0,0,0,0,0,0,0,0,0],[0,0,0,0,0,0,0]];
    TASK PERS trackdata track38:=[0,FALSE,50,[0,0,0,0,0,0,0,0,0],[0,0,0,0,0,0,0]];
    TASK PERS trackdata track39:=[0,FALSE,50,[0,0,0,0,0,0,0,0,0],[0,0,0,0,0,0,0]];
    TASK PERS trackdata track40:=[0,FALSE,50,[0,0,0,0,0,0,0,0,0],[0,0,0,0,0,0,0]];

    TASK VAR intnum inumMoveG_PosHold;

    PERS bool bGanTry_Last_pos;
    PERS bool bTouch_last_R1_Comp;
    PERS bool bTouch_last_R2_Comp;
    PERS bool bGanTry_First_pos;
    PERS bool bTouch_First_R1_Comp;
    PERS bool bTouch_First_R2_Comp;
    PERS num nMacro010{2}:=[4,4];
    PERS num nMacro001{2}:=[4,4];
    PERS bool bEndSearchComplete;
    PERS edgedata edgeStart{2}:=[[[18363.5,4423.9,4.92933],50,50,0,12,0,0],[[18363.9,4411.91,4.65171],50,50,0,12,0,0]];
    PERS edgedata edgeEnd{2}:=[[[19008.1,4446.95,5.66316],50,50,0,12,0,0],[[19008.5,4434.96,5.38554],50,50,0,12,0,0]];
    PERS corrorder corrStart{10}:=[[20,30,10,25,40,10,15,30,10,2],[20,30,10,25,40,10,15,30,10,0],[-15,-30,-10,25,40,10,15,30,10,2],[0,0,0,25,40,10,15,30,10,0],[0,0,0,25,40,20,15,30,20,0],[-15,-30,-10,25,40,10,15,30,10,0],[999,0,0,0,0,0,0,0,0,0],[999,0,0,0,0,0,0,0,0,0],[999,0,0,25,40,10,15,30,30,10],[999,0,0,0,0,0,0,0,0,0]];
    PERS corrorder corrEnd{10}:=[[20,30,10,25,40,10,15,30,10,2],[20,30,10,25,40,10,15,30,10,0],[-15,-30,-10,25,40,10,15,30,10,2],[0,0,0,25,40,10,15,30,10,0],[0,0,0,25,40,20,15,40,20,0],[-15,-30,-10,25,40,10,15,30,10,0],[999,0,0,25,40,10,15,30,10,0],[999,0,0,0,0,0,0,0,0,0],[0,0,0,25,40,10,15,30,10,0],[0,0,0,0,0,0,0,0,0,0]];
    PERS pos pCorredStartPos{2};
    PERS pos pCorredEndPos{2};

    PERS num nCorrX_Store_Start{2};
    PERS num nCorrY_Store_Start{2};
    PERS num nCorrZ_Store_Start{2};
    PERS num nCorrX_Store_End{2};
    PERS num nCorrY_Store_End{2};
    PERS num nCorrZ_Store_End{2};

    TASK PERS num nCorrFailOffs_Y:=0;
    TASK PERS num nCorrFailOffs_Z:=0;
    CONST bool bEnd:=FALSE;
    CONST bool bStart:=TRUE;


    PERS torchmotion macroStartBuffer2{10};
    PERS torchmotion macroEndBuffer2{10};
    PERS num nWeldLineLength:=400;
    ! 264.966;
    PERS num nWeldLineLength_R2;
    ! 264.966;
    PERS robtarget pSearchStart:=[[0,-37.0002,4.16317],[0.270598,-0.653282,-0.653282,-0.270598],[0,0,0,1],[9E+09,9E+09,9E+09,9E+09,9E+09,9E+09]];
    PERS robtarget pSearchEnd:=[[0,15,4.16317],[0.270598,-0.653282,-0.653282,-0.270598],[0,0,0,1],[9E+09,9E+09,9E+09,9E+09,9E+09,9E+09]];
    TASK PERS string TouchErrorDirSub:="Start_Y";
    TASK PERS string TouchErrorDirMain:="Ready";
    PERS num nTouchRetryCount{2};
    PERS num n_Angle;
    TASK PERS num RetryDepthData{3}:=[10,10,10];
    PERS robtarget pWeldPosR2{40}:=[[[-3,7,1],[0.307623,-0.549545,-0.742667,-0.227629],[-1,0,0,1],[-8704.03,-8704.03,294.161,1030.31,9E+09,9E+09]],[[-3,7,1],[0.307623,-0.549545,-0.742667,-0.227629],[-1,0,0,1],[-8704.03,-8704.03,294.161,1030.31,9E+09,9E+09]],[[-3,-4.5,1],[0.307623,-0.549545,-0.742667,-0.227629],[-1,0,0,1],[-8704.03,-8704.03,294.161,1030.31,9E+09,9E+09]],[[15,-1,1],[0.307623,-0.549545,-0.742667,-0.227629],[-1,0,0,1],[-8704.03,-8704.03,294.161,1030.34,9E+09,9E+09]],[[200,-1,1],[0.270598,-0.653282,-0.653282,-0.270598],[-1,0,0,1],[-8704.03,-8704.03,294.161,1030.72,9E+09,9E+09]],[[1390,-1.00592,0.996463],[0.270597,-0.653283,-0.653281,-0.270597],[0,0,-1,1],[-8707.81,-8707.8,1477.15,1033.13,9E+09,9E+09]],[[0,0,0],[0,0,0,0],[0,0,0,0],[0,0,0,0,0,0]],[[0,0,0],[0,0,0,0],[0,0,0,0],[0,0,0,0,0,0]],[[0,0,0],[0,0,0,0],[0,0,0,0],[0,0,0,0,0,0]],[[0,0,0],[0,0,0,0],[0,0,0,0],[0,0,0,0,0,0]],[[0,0,0],[0,0,0,0],[0,0,0,0],[0,0,0,0,0,0]],[[0,0,0],[0,0,0,0],[0,0,0,0],[0,0,0,0,0,0]],[[0,0,0],[0,0,0,0],[0,0,0,0],[0,0,0,0,0,0]],[[0,0,0],[0,0,0,0],[0,0,0,0],[0,0,0,0,0,0]],[[0,0,0],[0,0,0,0],[0,0,0,0],[0,0,0,0,0,0]],[[0,0,0],[0,0,0,0],[0,0,0,0],[0,0,0,0,0,0]],[[0,0,0],[0,0,0,0],[0,0,0,0],[0,0,0,0,0,0]],[[0,0,0],[0,0,0,0],[0,0,0,0],[0,0,0,0,0,0]],[[0,0,0],[0,0,0,0],[0,0,0,0],[0,0,0,0,0,0]],[[0,0,0],[0,0,0,0],[0,0,0,0],[0,0,0,0,0,0]],[[0,0,0],[0,0,0,0],[0,0,0,0],[0,0,0,0,0,0]],[[0,0,0],[0,0,0,0],[0,0,0,0],[0,0,0,0,0,0]],[[0,0,0],[0,0,0,0],[0,0,0,0],[0,0,0,0,0,0]],[[0,0,0],[0,0,0,0],[0,0,0,0],[0,0,0,0,0,0]],[[0,0,0],[0,0,0,0],[0,0,0,0],[0,0,0,0,0,0]],[[0,0,0],[0,0,0,0],[0,0,0,0],[0,0,0,0,0,0]],[[0,0,0],[0,0,0,0],[0,0,0,0],[0,0,0,0,0,0]],[[0,0,0],[0,0,0,0],[0,0,0,0],[0,0,0,0,0,0]],[[0,0,0],[0,0,0,0],[0,0,0,0],[0,0,0,0,0,0]],[[0,0,0],[0,0,0,0],[0,0,0,0],[0,0,0,0,0,0]],[[0,0,0],[0,0,0,0],[0,0,0,0],[0,0,0,0,0,0]],[[0,0,0],[0,0,0,0],[0,0,0,0],[0,0,0,0,0,0]],[[0,0,0],[0,0,0,0],[0,0,0,0],[0,0,0,0,0,0]],[[0,0,0],[0,0,0,0],[0,0,0,0],[0,0,0,0,0,0]],[[0,0,0],[0,0,0,0],[0,0,0,0],[0,0,0,0,0,0]],[[0,0,0],[0,0,0,0],[0,0,0,0],[0,0,0,0,0,0]],[[0,0,0],[0,0,0,0],[0,0,0,0],[0,0,0,0,0,0]],[[0,0,0],[0,0,0,0],[0,0,0,0],[0,0,0,0,0,0]],[[0,0,0],[0,0,0,0],[0,0,0,0],[0,0,0,0,0,0]],[[1390,-1,1],[0.270598,-0.653282,-0.653282,-0.270598],[-1,0,0,1],[-8707.8,-8707.8,1477.15,1033.12,9E+09,9E+09]]];
    PERS num nRobCorrSpaceHeight;
    PERS pos pCorredPosBuffer:=[-0.000742761,3.88479,5.49397];
    PERS bool bWireTouch2;
    CONST robtarget pNull:=[[0,0,0],[1,0,0,0],[0,0,0,0],[9E+09,9E+09,9E+09,9E+09,9E+09,9E+09]];

    PERS bool bRobSwap;
    PERS jointtarget jCorrT_ROB2_Start;
    PERS jointtarget jCorrT_ROB2_End;
    PERS robtarget pCorrT_ROB2_Start;
    PERS robtarget pCorrT_ROB2_End;

    !!!!jWireCut
    TASK PERS num nWireCutSpeed:=600;
    PERS tooldata tWeld2:=[TRUE,[[319.990,0,331.830],[0.92590,0,0.37784,0]],[3.1,[-71.4,3.8,173.2],[1,0,0,0],0.055,0.049,0.005]];
    PERS tooldata tWeld2copy:=[TRUE,[[320.377,0,330.247],[0.92587,0,0.37784,0]],[3.1,[-71.4,3.8,173.2],[1,0,0,0],0.055,0.049,0.005]];
    PERS bool bEnableWeldSkip;
    PERS num nTrapCheck_2:=0;
    PERS seamdata smDefault_2Trap;
    VAR num tool_rx_end{3};
    VAR num tool_rx_start{3};
    VAR num tool_rx_delta{3};
    VAR robtarget pcalcWeldpos;
    VAR robtarget pMoveWeldpos;
    VAR robtarget pSaveWeldpos;
    !Error
    TASK VAR intnum iErrorDuringEntry;
    PERS num nEntryRetryCount{2};
    TASK VAR intnum iMoveHome_RBT2;
    TASK PERS bool bTouchWorkCount{6}:=[FALSE,FALSE,FALSE,FALSE,FALSE,FALSE];
    PERS monRobs MonitorweldErrorpostion;
    PERS monRobs MonitorPosition;
    PERS pos posStart;
    PERS pos posEnd;
    PERS bool bGantryInTrap{2};
    TASK VAR intnum intOutGantryHold;
    PERS edgedata edgestartBuffer2;
    PERS edgedata edgeEndBuffer2;
    PERS num nStartThick;
    PERS num nEndThick;
    PERS bool bBreakPoint{2};
    PERS num nBreakPoint{2};
    PERS bool btouchTimeOut{2};
    PERS bool bWeldOutputDisable;
    TASK PERS seamdata tsm2:=[0.5,0.5,[0,0,32,0,0,380,0,0,0],0,0,0,0,0,[0,0,0,0,0,0,0,0,0],0,1,[0,0,32,0,0,380,0,0,0],0,0,[0,0,0,0,0,0,0,0,0],0];
    TASK PERS welddata twel2:=[0.01,0,[0,0,32,0,0,380,0,0,0],[0,0,0,0,0,0,0,0,0]];
    TASK PERS weavedata tweav2:=[1,2,2,2,0,0,0,0,0,0,0,0,0,0,0];
    TASK PERS bool bInstalldir:=FALSE;
    PERS num nMoveid;
    PERS bool bExitCycle:=FALSE;

    TRAP trapOutGantryHold
        IDelete intOutGantryHold;
        bGantryInTrap{2}:=FALSE;
        Reset intReHoldGantry_2;
        Holdwd1:=[Welds2{1}.cpm/6,0,[5,0,Welds2{1}.voltage,Welds2{1}.wfs,0,Welds2{1}.Current,0,0,0],[0,0,0,0,0,0,0,0,0]];
        Holdwd2:=[Welds2{2}.cpm/6,0,[5,0,Welds2{2}.voltage,Welds2{2}.wfs,0,Welds2{2}.Current,0,0,0],[0,0,0,0,0,0,0,0,0]];
        Holdwd3:=[Welds2{3}.cpm/6,0,[5,0,Welds2{3}.voltage,Welds2{3}.wfs,0,Welds2{3}.Current,0,0,0],[0,0,0,0,0,0,0,0,0]];
        Holdwd4:=[Welds2{4}.cpm/6,0,[5,0,Welds2{4}.voltage,Welds2{4}.wfs,0,Welds2{4}.Current,0,0,0],[0,0,0,0,0,0,0,0,0]];
        Holdwd5:=[Welds2{5}.cpm/6,0,[5,0,Welds2{5}.voltage,Welds2{5}.wfs,0,Welds2{5}.Current,0,0,0],[0,0,0,0,0,0,0,0,0]];
        Holdwd6:=[Welds2{6}.cpm/6,0,[5,0,Welds2{6}.voltage,Welds2{6}.wfs,0,Welds2{6}.Current,0,0,0],[0,0,0,0,0,0,0,0,0]];
        Holdwd7:=[Welds2{7}.cpm/6,0,[5,0,Welds2{7}.voltage,Welds2{7}.wfs,0,Welds2{7}.Current,0,0,0],[0,0,0,0,0,0,0,0,0]];
        Holdwd8:=[Welds2{8}.cpm/6,0,[5,0,Welds2{8}.voltage,Welds2{8}.wfs,0,Welds2{8}.Current,0,0,0],[0,0,0,0,0,0,0,0,0]];
        Holdwd9:=[Welds2{9}.cpm/6,0,[5,0,Welds2{9}.voltage,Welds2{9}.wfs,0,Welds2{9}.Current,0,0,0],[0,0,0,0,0,0,0,0,0]];
        Holdwd10:=[Welds2{10}.cpm/6,0,[5,0,Welds2{10}.voltage,Welds2{10}.wfs,0,Welds2{10}.Current,0,0,0],[0,0,0,0,0,0,0,0,0]];
        ArcRefresh;
    ENDTRAP

    TRAP trapMoveG_PosHold
        rTrapWeldMove;
    ENDTRAP

    TRAP trapErrorDuringEntry
        Set po34_EntryR2Error;
        IDelete iMoveHome_RBT2;
        rErrorDuringEntry;
    ENDTRAP

    TRAP trapMoveHome_RBT2
        VAR robtarget pTemp;
        IDelete iMoveHome_RBT2;
        StopMove;
        ClearPath;
        StartMove;
        pTemp:=CRobT(\TaskName:="T_ROB2"\Tool:=tWeld2\WObj:=wobjWeldLine2);
        MoveL RelTool(pTemp,0,0,-10),vTargetSpeed,z0,tWeld2\WObj:=wobjWeldLine2;
        bWeldOutputDisable:=TRUE;
        stReact{2}:="Error_Arc_Touch";
        WaitSyncTask Wait{80},taskGroup123;
        WaitUntil stReact{1}="Error_Arc_Touch" AND stReact{2}="Error_Arc_Touch";
        WaitSyncTask Wait{81},taskGroup123;
        WaitUntil stCommand="Error_Arc_Touch";
        stReact{2}:="";
        WaitUntil stCommand="";
        WaitSyncTask Wait{82},taskGroup123;
        ExitCycle;

    ENDTRAP

    PROC main()
        VAR num update_counter := 0;
        VAR iodev main_logfile;
        VAR num test_mode;
        VAR num wait_count := 0;  ! v1.9.17: Wait counter for shared_test_mode

        ! Open main process log (do this before config read)
        Open "HOME:/task2_main_process.txt", main_logfile \Write;
        Write main_logfile, "TASK2 Main Log (" + TASK2_VERSION + ") Date=" + CDate() + " Time=" + CTime();
        Write main_logfile, "Main entry reached";
        TPWrite "TASK2: main entered";

        ! v1.9.17: Wait for TASK1 to set shared_test_mode (max 5 seconds)
        TPWrite "TASK2: Waiting for TASK1 shared_test_mode...";
        Write main_logfile, "Waiting for shared_test_mode...";
        wait_count := 0;
        WHILE shared_test_mode = 0 AND wait_count < 50 DO
            WaitTime 0.1;
            wait_count := wait_count + 1;
        ENDWHILE
        test_mode := shared_test_mode;
        Write main_logfile, "TEST_MODE=" + NumToStr(test_mode, 0) + " (from TASK1)";
        TPWrite "TASK2: TEST_MODE=" + NumToStr(test_mode, 0);

        ! Initialize synchronization flag
        robot2_init_complete := FALSE;

        ! Initialize Robot2 position
        TPWrite "========================================";
        TPWrite "TASK2: Starting Robot2 initialization...";
        TPWrite "========================================";
        SetRobot2InitialPosition;
        TPWrite "TASK2: Robot2 initialization completed";
        Write main_logfile, "Step1 done (Robot2 init)";

        ! Set synchronization flag to signal TASK1 (after Step1)
        robot2_init_complete := TRUE;
        TPWrite "TASK2: Synchronization flag set (robot2_init_complete = TRUE)";
        Write main_logfile, "Flag set (Robot2 init)";

        IF test_mode = 2 THEN
            Write main_logfile, "Mode2 offset start";
            SetRobot2OffsetPosition;
            Write main_logfile, "Mode2 offset applied";

            ! v1.8.74: Wait for TASK1 to reset flags and set mode2_config_ready
            ! This prevents race condition where TASK2 sets flag before TASK1 resets it
            Write main_logfile, "Mode2: Waiting for config_ready before signaling...";
            TPWrite "TASK2: Waiting for config_ready...";
            WHILE NOT mode2_config_ready DO
                WaitTime 0.1;
            ENDWHILE
            Write main_logfile, "Mode2: config_ready=TRUE, now signaling initial offset done";

            ! Signal TASK1 that initial offset is done
            mode2_r2_initial_offset_done := TRUE;
            Write main_logfile, "Mode2: Initial offset done signal sent";

            ! v1.8.63: Monitor for reposition triggers
            Write main_logfile, "Mode2: Entering reposition monitor loop";
            TPWrite "TASK2: Monitoring for reposition triggers...";
            WHILE mode2_config_ready DO
                IF mode2_r2_reposition_trigger THEN
                    Write main_logfile, "Reposition trigger received";
                    SetRobot2OffsetPosition;
                    mode2_r2_reposition_done := TRUE;
                    Write main_logfile, "Reposition complete, done=TRUE";
                    ! Wait for trigger to be cleared
                    WHILE mode2_r2_reposition_trigger DO
                        WaitTime 0.05;
                    ENDWHILE
                    mode2_r2_reposition_done := FALSE;
                ENDIF
                WaitTime 0.05;
            ENDWHILE
            Write main_logfile, "Mode2: Exited reposition monitor (config_ready=FALSE)";
        ELSEIF test_mode = 3 THEN
            ! v1.9.17: Weld Sequence - call Robot2_WeldSequence
            Write main_logfile, "Weld Sequence mode (test_mode=3)";
            TPWrite "TASK2: Weld Sequence mode";
            Robot2_WeldSequence;
            Write main_logfile, "Weld Sequence completed";
        ELSEIF test_mode = 9 THEN
            ! v1.9.24: TestMenu mode - Monitor for Full Weld Sequence sync
            Write main_logfile, "TestMenu mode (test_mode=9) - Sync monitor enabled";
            TPWrite "TASK2: TestMenu mode - Weld sync monitoring";
            ! Monitor for weld sync signal from TASK1's TestFullWeldSequence (menu 11)
            WHILE TRUE DO
                IF t1_weld_position_ready = TRUE THEN
                    Write main_logfile, "Weld sync detected, running Robot2_EdgeWeldSequence";
                    TPWrite "TASK2: Weld sync detected, positioning Robot2...";
                    Robot2_EdgeWeldSequence;
                    Write main_logfile, "Robot2_EdgeWeldSequence completed";
                    TPWrite "TASK2: Sequence complete";
                    ! Wait for TASK1 to reset flag before next cycle
                    TPWrite "TASK2: Waiting for flag reset...";
                    WHILE t1_weld_position_ready = TRUE DO
                        WaitTime 0.1;
                    ENDWHILE
                    TPWrite "TASK2: Flag reset, ready for next cycle";
                    Write main_logfile, "Flag reset detected, resuming monitor";
                ENDIF
                WaitTime 0.2;
            ENDWHILE
        ELSEIF test_mode = 10 THEN
            ! v2.1.0: PlanA-style Command Loop
            Write main_logfile, "Command Loop mode (test_mode=10)";
            TPWrite "TASK2: Command Loop mode (PlanA Style)";
            Robot2_CommandLoop;
            Write main_logfile, "Command Loop exited";
        ELSEIF test_mode = 11 THEN
            ! v1.9.39: T_Head stCommand listener mode
            Write main_logfile, "T_Head Listener mode (test_mode=11)";
            TPWrite "TASK2: T_Head Listener mode";
            Rob2_CommandListener;
            Write main_logfile, "T_Head Listener exited";
        ENDIF

        WaitTime 1.0;

        ! Position update ready
        TPWrite "TASK2: Ready for cross-task measurement";
        Write main_logfile, "Ready for cross-task measurement";

        ! Close main log
        Write main_logfile, "TASK2 Main Process completed at " + CTime();
        Close main_logfile;

        TPWrite "========================================";
        TPWrite "TASK2: Initialization completed!";
        TPWrite "Check log files:";
        TPWrite "  - task2_main_process.txt";
        TPWrite "  - robot2_init_position.txt";
        TPWrite "========================================";

        ! Note: Position updates now handled by TASK1's UpdateRobot2BaseDynamicWobj
        ! No continuous loop needed - TASK1 reads Robot2 position on-demand
	ERROR
		TPWrite "ERROR in Rob2_MainModule main: " + NumToStr(ERRNO, 0);
		Close main_logfile;
		STOP;
    ENDPROC

    PROC rInit()
        AccSet 30,30;

        stReact{2}:="";
        WaitUntil stCommand="";
        stReact{2}:="Ready";
        IDelete inumMoveG_PosHold;
        IDelete iMoveHome_RBT2;
        IDelete intOutGantryHold;
        Reset intReHoldGantry_2;
        Reset soLn2Touch;
        bGantryInTrap{2}:=FALSE;
        RETURN ;
        MoveAbsJ [[0.0204923,-24.7246,-8.05237,0.0496605,-57.6256,1.6],[9E+09,9E+09,9E+09,9E+09,9E+09,9E+09]]\NoEOffs,v1000,z50,tool0;
        MoveJ [[168.50,0.00,1167.50],[0.999973,0.000344359,-0.00351527,0.00652012],[0,0,0,1],[9E+09,9E+09,9E+09,9E+09,9E+09,9E+09]],v1000,z50,tool0;
        RETURN ;
        ArcLStart [[-2.89,-0.02,1.95],[0.307559,-0.549626,-0.742627,-0.227649],[-1,-1,0,1],[9E+09,9E+09,9E+09,9E+09,9E+09,9E+09]],v10,smDefault_2{1},wd2,fine,tWeld2\WObj:=wobjWeldLine2;
        ArcLEnd [[31.01,-0.07,1.91],[0.307527,-0.549634,-0.742645,-0.227613],[-1,-1,0,1],[9E+09,9E+09,9E+09,9E+09,9E+09,9E+09]],v10,smDefault_2{1},wd2,fine,tWeld2\WObj:=wobjWeldLine2;
        RETURN ;
        MoveL [[0,0,0],[0.264906,0.659459,-0.649912,0.269356],[0,0,0,1],[9E+09,9E+09,9E+09,9E+09,9E+09,9E+09]],v10,z50,tWeld2\WObj:=wobjWeldLine2;
    ENDPROC

    !    PROC rTrapNoWeldMove()
    !        VAR num i;
    !        VAR targetdata WeldsTemp;
    !        VAR robtarget pWeldTemp;

    !        StopMove;
    !        StorePath;

    !        i:=nRunningStep{2};
    !        WeldsTemp:=Welds2{i};
    !        pWeldTemp:=CRobT(\taskname:="T_ROB2"\Tool:=tWeld2\WObj:=wobjWeldLine2);
    !        WeldsTemp.position:=pWeldTemp;
    !        ConfL\Off;
    !        While (so_MoveG_PosHold=1) DO
    !            nTrapCheck_2:=1;
    !            MoveL RelTool(WeldsTemp.position,0,-0.1,0),vWeld{i},fine,tWeld2\WObj:=wobjWeldLine2;
    !            MoveL RelTool(WeldsTemp.position,0,0.1,0),vWeld{i},fine,tWeld2\WObj:=wobjWeldLine2;
    !        ENDWHILE
    !        ConfL\On;
    !        RestoPath;
    !        StartMove;
    !    ENDPROC

    PROC rTrapWeldMove()
        VAR num i;
        VAR robtarget pWeldTemp;
        VAR robtarget pTemp_pos;
        VAR num nTempMmps;
        VAR speeddata vWeldTemp;
        IDelete inumMoveG_PosHold;
        StopMove;
        !        ClearPath;
        !        StorePath;
        i:=nRunningStep{2};
        nTempMmps:=Welds2{i}.cpm/6;
        vWeldTemp:=[nTempMmps,200,200,200];
        pWeldTemp:=CRobT(\taskname:="T_ROB2"\Tool:=tWeld2\WObj:=wobjWeldLine2);
        StartMove;
        ConfL\Off;
        WHILE (so_MoveG_PosHold=1) DO
            nTrapCheck_2:=2;
            MoveL Offs(pWeldTemp,0,0,0),vWeldTemp,fine,tWeld2\WObj:=wobjWeldLine2;
            MoveL Offs(pWeldTemp,0,0,0),vWeldTemp,fine,tWeld2\WObj:=wobjWeldLine2;
        ENDWHILE
        ConfL\On;
        !        RestoPath;

    ENDPROC

    PROC rMoveCorrConnect(num X,num Y,num Z,num Rx,num Ry,num Rz,num EAX_D,bool isStartPos,bool CCW,\switch LIN)
        VAR robtarget pTempConnect;
        VAR num nCorrX_Store;
        VAR num nCorrY_Store;
        VAR num nCorrZ_Store;

        IF (isStartPos=bStart) THEN
            nCorrX_Store:=nCorrX_Store_Start{2};
            nCorrY_Store:=nCorrY_Store_Start{2};
            nCorrZ_Store:=nCorrZ_Store_Start{2};
        ELSE
            nCorrX_Store:=nCorrX_Store_End{2};
            nCorrY_Store:=nCorrY_Store_End{2};
            nCorrZ_Store:=nCorrZ_Store_End{2};
        ENDIF


        pTempConnect:=pNull;
        pTempConnect.robconf:=[0,0,0,1];

        IF isStartPos=bStart THEN
            !        pTempConnect:=ConvertTcpToGantryCoord(pWeldPosR2{2}.position);
            IF CCW=FALSE THEN
                pTempConnect.trans:=[nCorrX_Store+(-1*X),nCorrY_Store+(Y),nCorrZ_Store+(Z)];
                pTempConnect.rot:=[0.5,-0.5,-0.5,-0.5];
                pTempConnect:=RelTool(pTempConnect,0,0,0\Rx:=macroStartBuffer2{1}.TravelAngle\Ry:=-1*macroStartBuffer2{1}.WorkingAngle+nBreakPoint{2});
            ELSE
                pTempConnect.trans:=[nCorrX_Store+(-1*X),nCorrY_Store+(Y*(-1)),nCorrZ_Store+(Z)];
                pTempConnect.rot:=[0.5,0.5,-0.5,0.5];
                pTempConnect:=RelTool(pTempConnect,0,0,0\Rx:=-1*macroStartBuffer2{1}.TravelAngle\Ry:=-1*macroStartBuffer2{1}.WorkingAngle+nBreakPoint{2});
            ENDIF
        ELSEIF isStartPos=bEnd THEN
            !        pTempConnect:=ConvertTcpToGantryCoord(pWeldPosR2{nMotionStepCount}.position);
            IF CCW=FALSE THEN
                pTempConnect.trans:=[nWeldLineLength_R2+nCorrX_Store+(X),nCorrY_Store+(Y),nCorrZ_Store+(Z)];
                pTempConnect.rot:=[0.5,-0.5,-0.5,-0.5];
                pTempConnect:=RelTool(pTempConnect,0,0,0\Rx:=macroEndBuffer2{nMotionEndStepLast{2}}.TravelAngle\Ry:=-1*macroEndBuffer2{nMotionEndStepLast{2}}.WorkingAngle+nBreakPoint{2});
            ELSE
                pTempConnect.trans:=[nWeldLineLength_R2+nCorrX_Store+(X),nCorrY_Store+(Y*(-1)),nCorrZ_Store+(Z)];
                pTempConnect.rot:=[0.5,0.5,-0.5,0.5];
                pTempConnect:=RelTool(pTempConnect,0,0,0\Rx:=-1*macroEndBuffer2{nMotionEndStepLast{2}}.TravelAngle\Ry:=-1*macroEndBuffer2{nMotionEndStepLast{2}}.WorkingAngle+nBreakPoint{2});
            ENDIF
        ENDIF

        IF Present(LIN)=FALSE THEN
            MoveJ pTempConnect,v300,fine,tWeld2\WObj:=wobjWeldLine2;
        ELSE
            MoveL pTempConnect,v300,fine,tWeld2\WObj:=wobjWeldLine2;
        ENDIF

        RETURN ;
    ENDPROC

    PROC rCorrSearchWeldLineEdgeX(num X,num Y,num Z,num Depth,num RetX,bool isStartPos,bool CCW,string dirErrorCheck)
        VAR num nCorrX_Store;
        VAR num nCorrY_Store;
        VAR num nCorrZ_Store;
        WaitUntil bRobSwap=CCW;
        IF (isStartPos=bStart) THEN
            nCorrX_Store:=nCorrX_Store_Start{2};
            nCorrY_Store:=nCorrY_Store_Start{2};
            nCorrZ_Store:=nCorrZ_Store_Start{2};
        ELSE
            nCorrX_Store:=nCorrX_Store_End{2};
            nCorrY_Store:=nCorrY_Store_End{2};
            nCorrZ_Store:=nCorrZ_Store_End{2};
        ENDIF

        TouchErrorDirSub:=dirErrorCheck;
        IF TouchErrorDirMain=dirErrorCheck AND nTouchRetryCount{2}>0 THEN
            IF (isStartPos=bEnd AND (nMacro001{1}=2 OR nMacro001{1}=5)) OR (isStartPos=bStart AND (nMacro010{1}=2 OR nMacro010{1}=5)) THEN
                Depth:=Depth+((RetryDepthData{1}*(-1))*nTouchRetryCount{2});
            ELSE
                Depth:=Depth+(RetryDepthData{1}*nTouchRetryCount{2});
            ENDIF
        ENDIF
        !!! Search weld X edge !!!
        WaitUntil bRobSwap=CCW;
        IF (isStartPos=bStart) THEN
            !        pSearchStart:=ConvertTcpToGantryCoord(pWeldPosR2{1}.position);
            pSearchStart.rot:=Welds2{1}.position.rot;
            IF (CCW=FALSE) pSearchStart.trans:=[nCorrX_Store+(-1*X),nCorrY_Store+(Y),nCorrZ_Store+(Z)];
            IF (CCW=TRUE) pSearchStart.trans:=[nCorrX_Store+(-1*X),nCorrY_Store+(Y*(-1)),nCorrZ_Store+(Z)];
        ELSEIF (isStartPos=bEnd) THEN
            !        pSearchStart:=ConvertTcpToGantryCoord(pWeldPosR2{nMotionStepCount}.position);
            !  pSearchStart.rot:=pWeldPosR2{nMotionStepCount{2}}.rot;
            pSearchStart.rot:=Welds2{nMotionStepCount{2}}.position.rot;
            IF (CCW=FALSE) pSearchStart.trans:=[nWeldLineLength_R2+nCorrX_Store+(X),nCorrY_Store+(Y),nCorrZ_Store+(Z)];
            IF (CCW=TRUE) pSearchStart.trans:=[nWeldLineLength_R2+nCorrX_Store+(X),nCorrY_Store+(Y*(-1)),nCorrZ_Store+(Z)];
        ENDIF

        pSearchStart.robconf.cfx:=1;
        pSearchStart.extax:=[9e9,9e9,9e9,9e9,9e9,9e9];
        !    pSearchStart.extax.eax_d:=wobjWeldLine1.uframe.trans.z-(nRobCorrSpaceHeight+wobjWeldLine1.oframe.trans.z);

        pSearchEnd:=pSearchStart;
        IF (isStartPos=bStart) pSearchEnd.trans.x:=pSearchStart.trans.x+Depth;
        IF (isStartPos=bEnd) pSearchEnd.trans.x:=pSearchStart.trans.x-Depth;

        rCorrSearchByWire pSearchStart,pSearchEnd\X;

        IF (isStartPos=bStart) nCorrX_Store:=pCorredPosBuffer.x;
        IF (isStartPos=bEnd) nCorrX_Store:=pCorredPosBuffer.x-nWeldLineLength_R2;

        IF (isStartPos=bStart) THEN
            nCorrX_Store_Start{2}:=nCorrX_Store;
            nCorrY_Store_Start{2}:=nCorrY_Store;
            nCorrZ_Store_Start{2}:=nCorrZ_Store;
        ELSE
            nCorrX_Store_End{2}:=nCorrX_Store;
            nCorrY_Store_End{2}:=nCorrY_Store;
            nCorrZ_Store_End{2}:=nCorrZ_Store;
        ENDIF

        rMoveCorrConnect RetX,Y,Z,0,0,0,pSearchStart.extax.eax_d,isStartPos,CCW;
        nTouchRetryCount{2}:=0;
        TouchErrorDirMain:="Ready";

        RETURN ;
    ENDPROC

    PROC rCorrSearchWeldLineEdgeY(num X,num Y,num Z,num Depth,num RetY,bool isStartPos,bool CCW,string dirErrorCheck)
        VAR num nCorrX_Store;
        VAR num nCorrY_Store;
        VAR num nCorrZ_Store;
        WaitUntil bRobSwap=CCW;
        IF (isStartPos=bStart) THEN
            nCorrX_Store:=nCorrX_Store_Start{2};
            nCorrY_Store:=nCorrY_Store_Start{2};
            nCorrZ_Store:=nCorrZ_Store_Start{2};
        ELSE
            nCorrX_Store:=nCorrX_Store_End{2};
            nCorrY_Store:=nCorrY_Store_End{2};
            nCorrZ_Store:=nCorrZ_Store_End{2};
        ENDIF

        TouchErrorDirSub:=dirErrorCheck;
        RetryDepthData{2}:=RetryDepthData{2}*(-1);
        IF TouchErrorDirMain=dirErrorCheck AND nTouchRetryCount{2}>0 Depth:=Depth+(RetryDepthData{2}*nTouchRetryCount{2});
        RetryDepthData{2}:=RetryDepthData{2}*(-1);

        !!! Search weld Y edge !!!
        WaitUntil bRobSwap=CCW;
        IF (isStartPos=bStart) THEN
            !        pSearchStart:=ConvertTcpToGantryCoord(pWeldPosR2{1}.position);
            pSearchStart.rot:=Welds2{1}.position.rot;
            IF (CCW=FALSE) pSearchStart.trans:=[nCorrX_Store+(-1*X),nCorrY_Store+(Y),nCorrZ_Store+(Z)];
            IF (CCW=TRUE) pSearchStart.trans:=[nCorrX_Store+(-1*X),nCorrY_Store+(Y*(-1)),nCorrZ_Store+Z];
        ELSEIF (isStartPos=bEnd) THEN
            !        pSearchStart:=ConvertTcpToGantryCoord(pWeldPosR2{nMotionStepCount}.position);
            !pSearchStart.rot:=pWeldPosR2{nMotionStepCount{2}}.rot;
            pSearchStart.rot:=Welds2{nMotionStepCount{2}}.position.rot;
            IF (CCW=FALSE) pSearchStart.trans:=[nWeldLineLength_R2+nCorrX_Store+(X),nCorrY_Store+(Y),nCorrZ_Store+(Z)];
            IF (CCW=TRUE) pSearchStart.trans:=[nWeldLineLength_R2+nCorrX_Store+(X),nCorrY_Store+(Y*(-1)),nCorrZ_Store+(Z)];
        ENDIF

        pSearchStart.robconf.cfx:=1;
        !  pSearchStart.extax.eax_d:=wobjWeldLine1.uframe.trans.z-(nRobCorrSpaceHeight+wobjWeldLine1.oframe.trans.z);

        pSearchEnd:=pSearchStart;
        pSearchStart.extax:=[9e9,9e9,9e9,9e9,9e9,9e9];
        IF (CCW=FALSE) pSearchEnd.trans.y:=pSearchStart.trans.y-Depth;
        IF (CCW=TRUE) pSearchEnd.trans.y:=pSearchStart.trans.y+Depth;

        rCorrSearchByWire pSearchStart,pSearchEnd\Y;

        nCorrY_Store:=pCorredPosBuffer.y;

        IF (isStartPos=bStart) THEN
            nCorrX_Store_Start{2}:=nCorrX_Store;
            nCorrY_Store_Start{2}:=nCorrY_Store;
            nCorrZ_Store_Start{2}:=nCorrZ_Store;
        ELSE
            nCorrX_Store_End{2}:=nCorrX_Store;
            nCorrY_Store_End{2}:=nCorrY_Store;
            nCorrZ_Store_End{2}:=nCorrZ_Store;
        ENDIF

        rMoveCorrConnect X,RetY,Z,0,0,0,pSearchStart.extax.eax_d,isStartPos,CCW;
        nTouchRetryCount{2}:=0;
        TouchErrorDirMain:="Ready";

        RETURN ;
    ENDPROC

    PROC rCorrSearchWeldLineEdgeZ(num X,num Y,num Z,num Depth,num RetZ,bool isStartPos,bool CCW,string dirErrorCheck)
        VAR num nCorrX_Store;
        VAR num nCorrY_Store;
        VAR num nCorrZ_Store;
        WaitUntil bRobSwap=CCW;
        IF (isStartPos=bStart) THEN
            nCorrX_Store:=nCorrX_Store_Start{2};
            nCorrY_Store:=nCorrY_Store_Start{2};
            nCorrZ_Store:=nCorrZ_Store_Start{2};
        ELSE
            nCorrX_Store:=nCorrX_Store_End{2};
            nCorrY_Store:=nCorrY_Store_End{2};
            nCorrZ_Store:=nCorrZ_Store_End{2};
        ENDIF
        TouchErrorDirSub:=dirErrorCheck;
        IF TouchErrorDirMain=dirErrorCheck AND nTouchRetryCount{2}>0 Depth:=Depth+(RetryDepthData{3}*nTouchRetryCount{2});
        !!! Search weld Z edge !!!
        WaitUntil bRobSwap=CCW;
        IF (isStartPos=bStart) THEN
            !       pSearchStart:=ConvertTcpToGantryCoord(pWeldPosR2{1}.position);
            pSearchStart.rot:=Welds2{1}.position.rot;
            IF (CCW=FALSE) pSearchStart.trans:=[nCorrX_Store+(-1*X),nCorrY_Store+(Y),nCorrZ_Store+(Z)];
            IF (CCW=TRUE) pSearchStart.trans:=[nCorrX_Store+(-1*X),nCorrY_Store+(Y*(-1)),nCorrZ_Store+(Z)];
        ELSEIF (isStartPos=bEnd) THEN
            !        pSearchStart:=ConvertTcpToGantryCoord(pWeldPosR2{nMotionStepCount}.position);
            pSearchStart.rot:=Welds2{nMotionStepCount{2}}.position.rot;
            ! pSearchStart.rot:=pWeldPosR2{nMotionStepCount{2}}.rot;
            IF (CCW=FALSE) pSearchStart.trans:=[nWeldLineLength_R2+nCorrX_Store+(X),nCorrY_Store+(Y),nCorrZ_Store+(Z)];
            IF (CCW=TRUE) pSearchStart.trans:=[nWeldLineLength_R2+nCorrX_Store+(X),nCorrY_Store+(Y*(-1)),nCorrZ_Store+(Z)];
        ENDIF

        pSearchStart.robconf.cfx:=1;
        pSearchStart.extax:=[9e9,9e9,9e9,9e9,9e9,9e9];
        !  pSearchStart.extax.eax_d:=wobjWeldLine1.uframe.trans.z-(nRobCorrSpaceHeight+wobjWeldLine1.oframe.trans.z);

        pSearchEnd:=pSearchStart;
        pSearchEnd.trans.z:=pSearchStart.trans.z-Depth;

        rCorrSearchByWire pSearchStart,pSearchEnd\Z;

        nCorrZ_Store:=pCorredPosBuffer.z;

        IF (isStartPos=bStart) THEN
            nCorrX_Store_Start{2}:=nCorrX_Store;
            nCorrY_Store_Start{2}:=nCorrY_Store;
            nCorrZ_Store_Start{2}:=nCorrZ_Store;
        ELSE
            nCorrX_Store_End{2}:=nCorrX_Store;
            nCorrY_Store_End{2}:=nCorrY_Store;
            nCorrZ_Store_End{2}:=nCorrZ_Store;
        ENDIF

        rMoveCorrConnect X,Y,RetZ,0,0,0,pSearchStart.extax.eax_d,isStartPos,CCW;
        nTouchRetryCount{2}:=0;
        TouchErrorDirMain:="Ready";

        RETURN ;
    ENDPROC

    PROC rCorrSearchByWire(robtarget SearchStart,robtarget SearchEnd,\switch X\switch Y\switch Z)
        VAR robtarget pTemp:=[[0,0,0],[1,0,0,0],[0,0,0,0],[0,0,0,0,9E+09,9E+09]];
        MoveJ SearchStart,v100,fine,tWeld2\WObj:=wobjWeldLine2;
        rCheckWelder;
        SearchL\SStop,bWireTouch2,SearchStart,SearchEnd,v10,tWeld2\WObj:=wobjWeldLine2;

        Reset soLn2Touch;
        WaitTime 0;
        WaitUntil(siLn2TouchActive=0);
        pTemp:=CRobT(\taskname:="T_ROB2"\tool:=tWeld2\WObj:=wobjWeldLine2);
        pCorredPosBuffer:=pTemp.trans;
        !        stop;
        RETURN ;
    ERROR

        TouchErrorDirMain:=TouchErrorDirSub;
        IDelete iMoveHome_RBT2;
        IF ERRNO=ERR_WHLSEARCH THEN
            rTouchErrorHandling 2;
        ELSEIF ERRNO=ERR_SIGSUPSEARCH THEN
            WaitTime 999;
            rTouchErrorHandling 3;
        ELSE
            rTouchErrorHandling 3;
        ENDIF
    ENDPROC

    PROC rZero()
        MoveAbsJ [[0,0,0,0,0,0],[9E+09,9E+09,9E+09,9E+09,9E+09,9E+09]]\NoEOffs,v1000,fine,tool0;
    ENDPROC

    PROC rErrorDuringEntry()
        VAR robtarget pTemp;
        Reset soLn2Touch;
        StopMove;
        ClearPath;
        StartMove;
        pTemp:=CRobT(\TaskName:="T_ROB2"\Tool:=tWeld2\WObj:=wobjWeldLine2);
        MoveL RelTool(pTemp,0,0,-10),vTargetSpeed,fine,tWeld2\WObj:=wobjWeldLine2;
        stReact{2}:="Error_Arc_Touch";
        WaitSyncTask Wait{80},taskGroup123;
        WaitUntil stReact{1}="Error_Arc_Touch" AND stReact{2}="Error_Arc_Touch";
        WaitSyncTask Wait{81},taskGroup123;
        WaitUntil stCommand="Error_Arc_Touch";
        stReact{2}:="";
        WaitUntil stCommand="";
        WaitSyncTask Wait{82},taskGroup123;

        ExitCycle;
    ENDPROC

    PROC rArcError()
        VAR robtarget pTemp;

        IDelete iMoveHome_RBT2;
        StopMove;
        ClearPath;
        StartMove;
        IF bRobSwap=FALSE THEN
            Set po37_ArcR2Error;
            MonitorweldErrorpostion.monPose1:=MonitorPosition.monPose1;
            MonitorweldErrorpostion.monPose2:=MonitorPosition.monPose2;
        ELSE
            Set po36_ArcR1Error;
            MonitorweldErrorpostion.monPose1:=MonitorPosition.monPose1;
            MonitorweldErrorpostion.monPose2:=MonitorPosition.monPose2;
        ENDIF

        pTemp:=CRobT(\TaskName:="T_ROB2"\Tool:=tWeld2\WObj:=wobjWeldLine2);
        MoveL RelTool(pTemp,0,0,-10),vTargetSpeed,z0,tWeld2\WObj:=wobjWeldLine2;

        stReact{2}:="Error_Arc_Touch";
        WaitSyncTask Wait{80},taskGroup123;
        WaitUntil stReact{1}="Error_Arc_Touch" AND stReact{2}="Error_Arc_Touch";
        WaitSyncTask Wait{81},taskGroup123;
        WaitUntil stCommand="Error_Arc_Touch";
        stReact{2}:="";
        WaitUntil stCommand="";
        WaitSyncTask Wait{82},taskGroup123;
        ExitCycle;

    ENDPROC

    PROC rTouchErrorHandling(num Errorno)
        VAR robtarget pTemp;
        Reset soLn2Touch;
        Set po35_TouchR2Error;
        IDelete iMoveHome_RBT2;

        pTemp:=CRobT(\TaskName:="T_ROB2"\tool:=tWeld2\WObj:=wobjWeldLine2);
        MoveL RelTool(pTemp,0,0,-10),v200,z10,tWeld2\WObj:=wobjWeldLine2;
        stReact{2}:="Error_Arc_Touch";
        WaitSyncTask Wait{80},taskGroup123;
        WaitUntil stReact{1}="Error_Arc_Touch" AND stReact{2}="Error_Arc_Touch";
        WaitSyncTask Wait{81},taskGroup123;
        WaitUntil stCommand="Error_Arc_Touch";
        stReact{2}:="";
        WaitUntil stCommand="";
        WaitSyncTask Wait{82},taskGroup123;
        StartMove;
        ExitCycle;


    ENDPROC

    PROC rT_ROB2check()
        VAR robtarget pTemp;
        pTemp:=CRobT(\TaskName:="T_ROB2"\Tool:=tWeld2\WObj:=wobjWeldLine2);
        IF Abs(pTemp.trans.Y)<100 AND Abs(pTemp.trans.Z)<200 THEN
            IF pTemp.trans.Y>0 then
                pTemp.trans.y:=140;
                MoveL pTemp,v100,z10,tWeld2\WObj:=wobjWeldLine2;
            ENDIF
            IF pTemp.trans.Y<0 THEN
                pTemp.trans.y:=-140;
                MoveL pTemp,v100,z10,tWeld2\WObj:=wobjWeldLine2;
            ENDIF
        ENDIF
    ENDPROC

    PROC rCheckWelder()
        IF (soLn2Touch=1) THEN
            Reset soLn2Touch;
            WaitTime 0.5;
        ENDIF
        WaitTime 0.5;
        WaitUntil(siLn2TouchActive=0 OR soLn2Touch=0);
        Set soLn2Touch;
        WaitUntil(siLn2TouchActive=1 AND soLn2Touch=1);
    ENDPROC

    PROC rWeldinit()
        return1:
        !!!===ArcWareReset===!!!
        reset soAwDeleteSDB2;
        WaitUntil soAwDeleteSDB2=0\MaxTime:=5;
        reset soAwError2;
        WaitUntil soAwError2=0\MaxTime:=5;
        reset soAwGasOn2;
        WaitUntil soAwGasOn2=0\MaxTime:=5;
        reset soAwInitSDB2;
        WaitUntil soAwInitSDB2=0\MaxTime:=5;
        reset soAwManFeed15mm2;
        WaitUntil soAwManFeed15mm2=0\MaxTime:=5;
        reset soAwManFeedRev2;
        WaitUntil soAwManFeedRev2=0\MaxTime:=5;
        reset soAwManGasOn2;
        WaitUntil soAwManGasOn2=0\MaxTime:=5;
        reset soAwOnFlag2;
        WaitUntil soAwOnFlag2=0\MaxTime:=5;
        reset soAwRestart2;
        WaitUntil soAwRestart2=0\MaxTime:=5;
        reset soAwRunning2;
        WaitUntil soAwRunning2=0\MaxTime:=5;
        reset soAwWeldUpdate2;
        WaitUntil soAwWeldUpdate2=0\MaxTime:=5;
        set soAwTaskReady2;
        WaitUntil soAwTaskReady2=1\MaxTime:=5;
        set soAwStart2;
        WaitUntil soAwStart2=1\MaxTime:=5;
        set soAwEquipOK2;
        WaitUntil soAwEquipOK2=1\MaxTime:=5;
        !!!!!!!====Lincoln_Reset====!!!!
        reset soLn2AdjWireStickOut;
        WaitUntil soLn2AdjWireStickOut=0\MaxTime:=5;
        reset soLn2ArcOkLatch;
        WaitUntil soLn2ArcOkLatch=0\MaxTime:=5;
        set soLn2BusAvailable;
        WaitUntil soLn2BusAvailable=1\MaxTime:=5;
        reset soLn2EvalWeldDataLog;
        WaitUntil soLn2EvalWeldDataLog=0\MaxTime:=5;
        reset soLn2FeedOn;
        WaitUntil soLn2FeedOn=0\MaxTime:=5;
        reset soLn2Gas;
        WaitUntil soLn2Gas=0\MaxTime:=5;
        reset soLn2GasError;
        WaitUntil soLn2GasError=0\MaxTime:=5;
        set soLn2Installed;
        WaitUntil soLn2Installed=1\MaxTime:=5;
        set soLn2Listen;
        WaitUntil soLn2Listen=1\MaxTime:=5;
        reset soLn2LoadWeldModes;
        WaitUntil soLn2LoadWeldModes=0\MaxTime:=5;
        reset soLn2ManWireFeed;
        WaitUntil soLn2ManWireFeed=0\MaxTime:=5;
        set soLn2NOP_Enable;
        WaitUntil soLn2NOP_Enable=1\MaxTime:=5;
        reset soLn2NOPDisable;
        WaitUntil soLn2NOPDisable=0\MaxTime:=5;
        reset soLn2SaveCapLog;
        WaitUntil soLn2SaveCapLog=0\MaxTime:=5;
        reset soLn2ShowRecMessage;
        WaitUntil soLn2ShowRecMessage=0\MaxTime:=5;
        reset soLn2StartPart;
        WaitUntil soLn2StartPart=0\MaxTime:=5;
        set soLn2StartupComplete;
        WaitUntil soLn2StartupComplete=1\MaxTime:=5;
        reset soLn2StopProc;
        WaitUntil soLn2StopProc=0\MaxTime:=5;
        set soLn2T1Exec;
        WaitUntil soLn2T1Exec=1\MaxTime:=5;
        set soLn2T2Exec;
        WaitUntil soLn2T2Exec=1\MaxTime:=5;
        reset soLn2Touch;
        WaitUntil soLn2Touch=0\MaxTime:=5;
        reset soLn2TouchActive;
        WaitUntil soLn2TouchActive=0\MaxTime:=5;
        set soLn2ValidSchedule;
        WaitUntil soLn2ValidSchedule=1\MaxTime:=5;
        reset soLn2VoltError;
        WaitUntil soLn2VoltError=0\MaxTime:=5;
        reset soLn2WaterError;
        WaitUntil soLn2WaterError=0\MaxTime:=5;
        reset soLn2Weld;
        WaitUntil soLn2Weld=0\MaxTime:=5;
        reset soLn2WeldDataLogOn;
        WaitUntil soLn2WeldDataLogOn=0\MaxTime:=5;
        set soLn2WelderRdyDO;
        WaitUntil soLn2WelderRdyDO=1\MaxTime:=5;
        reset soLn2WeldError;
        WaitUntil soLn2WeldError=0\MaxTime:=5;
        reset soLn2WireBurnOff;
        WaitUntil soLn2WireBurnOff=0\MaxTime:=5;
        reset soLn2WireFeedError;
        WaitUntil soLn2WireFeedError=0\MaxTime:=5;
        set soLn2WireFeedRdyDO;
        WaitUntil soLn2WireFeedRdyDO=1\MaxTime:=5;
        reset soLn2WireStickDO;
        WaitUntil soLn2WireStickDO=0\MaxTime:=5;
        RETURN ;
        GOTO return1;
    ENDPROC

    PROC Routine2()
        MoveJ [[-0.00,981.00,441.10],[0.5,-0.5,0.5,0.5],[1,0,0,2],[9E+9,9E+9,9E+9,9E+9,9E+9,9E+9]],v1000,z50,tool0;
    ENDPROC

    PROC rUpdateR2Position()
        VAR num X;
        VAR num Y;
        VAR num Z;
        VAR num R;
        VAR num X2;
        VAR num Y2;
        VAR num Z2;
        !        jTemp:=[[0,0,0,0,0,0],[0,0,0,30,0,0]];
        jTemp := CJointT(\TaskName:="T_ROB1");

        X:=jtemp.extax.eax_a;
        Y:=jtemp.extax.eax_b;
        Z:=jtemp.extax.eax_c;
        R:=jtemp.extax.eax_d;

        X2:=X-(488*cos(R));
        !X2:=X-(976*cos(R));
        Y2:=Y-(488*sin(R));
        !Y2:=Y-(976*sin(R));

        nCaledR2Pos:=[X2,Y2,Z];
        wobjtest:=[FALSE,TRUE,"GantryRob",[[X2,Y2,Z],[1,0,0,0]],[[0,0,0],[1,0,0,0]]];

        ! Update Robot2 Floor position for cross-task measurement (v1.7.38)
        UpdateRobot2FloorPosition;
    ENDPROC

	!========================================
	! Robot2 Capability Tests
	!========================================
	! Version: v1.0.0
	! Date: 2025-12-17
	! Purpose: Verify Robot2 gantry external axis access

	!========================================
	! Test 1: Read External Axes via CJointT()
	!========================================
	PROC TestRobot2_ReadExternalAxes()
		VAR jointtarget current_joint;
		VAR num gantry_x;
		VAR num gantry_y;
		VAR num gantry_z;
		VAR num gantry_r;
		VAR num gantry_x2;
		VAR iodev logfile;

		TPWrite "========================================";
		TPWrite "Test 1: Robot2 - Read External Axes";
		TPWrite "========================================";

		current_joint := CJointT();

		TPWrite "Robot Joints:";
		TPWrite "  J1 = " + NumToStr(current_joint.robax.rax_1, 2) + " deg";
		TPWrite "  J2 = " + NumToStr(current_joint.robax.rax_2, 2) + " deg";
		TPWrite "  J3 = " + NumToStr(current_joint.robax.rax_3, 2) + " deg";
		TPWrite "  J4 = " + NumToStr(current_joint.robax.rax_4, 2) + " deg";
		TPWrite "  J5 = " + NumToStr(current_joint.robax.rax_5, 2) + " deg";
		TPWrite "  J6 = " + NumToStr(current_joint.robax.rax_6, 2) + " deg";

		gantry_x := current_joint.extax.eax_a;
		gantry_y := current_joint.extax.eax_b;
		gantry_z := current_joint.extax.eax_c;
		gantry_r := current_joint.extax.eax_d;
		gantry_x2 := current_joint.extax.eax_f;

		TPWrite "Gantry External Axes:";
		TPWrite "  X1 = " + NumToStr(gantry_x, 4) + " m";
		TPWrite "  Y  = " + NumToStr(gantry_y, 4) + " m";
		TPWrite "  Z  = " + NumToStr(gantry_z, 4) + " m";
		TPWrite "  R  = " + NumToStr(gantry_r, 4) + " rad";
		TPWrite "  X2 = " + NumToStr(gantry_x2, 4) + " m";

			Open "HOME:/robot2_external_axes_test.txt", logfile \Append;

		Write logfile, "========================================";
		Write logfile, "Robot2 - External Axes Reading Test";
		Write logfile, "========================================";
		Write logfile, "Date: " + CDate();
		Write logfile, "Time: " + CTime();
		Write logfile, "";
		Write logfile, "Robot Joints: ["
			+ NumToStr(current_joint.robax.rax_1, 2) + ", "
			+ NumToStr(current_joint.robax.rax_2, 2) + ", "
			+ NumToStr(current_joint.robax.rax_3, 2) + ", "
			+ NumToStr(current_joint.robax.rax_4, 2) + ", "
			+ NumToStr(current_joint.robax.rax_5, 2) + ", "
			+ NumToStr(current_joint.robax.rax_6, 2) + "]";
		Write logfile, "";
		Write logfile, "Gantry External Axes:";
		Write logfile, "  X1 = " + NumToStr(gantry_x, 4) + " m";
		Write logfile, "  Y  = " + NumToStr(gantry_y, 4) + " m";
		Write logfile, "  Z  = " + NumToStr(gantry_z, 4) + " m";
		Write logfile, "  R  = " + NumToStr(gantry_r, 4) + " rad";
		Write logfile, "  X2 = " + NumToStr(gantry_x2, 4) + " m";
		Write logfile, "";
		Write logfile, "Result: ";

		IF gantry_x <> 9E9 OR gantry_y <> 9E9 OR gantry_z <> 9E9 THEN
			Write logfile, "SUCCESS - Robot2 can read gantry external axes!";
			TPWrite "Result: SUCCESS";
		ELSE
			Write logfile, "FAIL - Robot2 cannot read gantry external axes";
			TPWrite "Result: FAIL";
		ENDIF

		Write logfile, "========================================\0A";
		Close logfile;

		TPWrite "========================================";
		TPWrite "Test 1 Complete. Check robot2_external_axes_test.txt";

	ERROR
		TPWrite "ERROR in TestRobot2_ReadExternalAxes: " + NumToStr(ERRNO, 0);
		Close logfile;
		TRYNEXT;
	ENDPROC

	!========================================
	! Test 2: Robot2 TCP Coordinates
	!========================================
	PROC TestRobot2_TCPCoordinates()
		VAR robtarget tcp_world;
		VAR robtarget tcp_wobj0;
		VAR robtarget tcp_base;
		VAR iodev logfile;

		TPWrite "========================================";
		TPWrite "Test 2: Robot2 - TCP Coordinates";
		TPWrite "========================================";

		tcp_world := CRobT(\Tool:=tool0);
		tcp_wobj0 := CRobT(\Tool:=tool0\WObj:=wobj0);
		tcp_base := tcp_wobj0;

		TPWrite "World Coordinates:";
		TPWrite "  X = " + NumToStr(tcp_world.trans.x, 3) + " mm";
		TPWrite "  Y = " + NumToStr(tcp_world.trans.y, 3) + " mm";
		TPWrite "  Z = " + NumToStr(tcp_world.trans.z, 3) + " mm";

		TPWrite "wobj0 Coordinates:";
		TPWrite "  X = " + NumToStr(tcp_wobj0.trans.x, 3) + " mm";
		TPWrite "  Y = " + NumToStr(tcp_wobj0.trans.y, 3) + " mm";
		TPWrite "  Z = " + NumToStr(tcp_wobj0.trans.z, 3) + " mm";

			Open "HOME:/robot2_tcp_coordinates.txt", logfile \Append;

		Write logfile, "========================================";
		Write logfile, "Robot2 - TCP Coordinates Test";
		Write logfile, "========================================";
		Write logfile, "Date: " + CDate();
		Write logfile, "Time: " + CTime();
		Write logfile, "";
		Write logfile, "1. World Coordinates:";
		Write logfile, "   X = " + NumToStr(tcp_world.trans.x, 3) + " mm";
		Write logfile, "   Y = " + NumToStr(tcp_world.trans.y, 3) + " mm";
		Write logfile, "   Z = " + NumToStr(tcp_world.trans.z, 3) + " mm";
		Write logfile, "";
		Write logfile, "2. wobj0 Coordinates:";
		Write logfile, "   X = " + NumToStr(tcp_wobj0.trans.x, 3) + " mm";
		Write logfile, "   Y = " + NumToStr(tcp_wobj0.trans.y, 3) + " mm";
		Write logfile, "   Z = " + NumToStr(tcp_wobj0.trans.z, 3) + " mm";
		Write logfile, "";
		Write logfile, "Note: Robot2 wobj0 should be at Robot2 Base";
		Write logfile, "========================================\0A";

		Close logfile;

		TPWrite "========================================";
		TPWrite "Test 2 Complete. Check robot2_tcp_coordinates.txt";

	ERROR
		TPWrite "ERROR in TestRobot2_TCPCoordinates: " + NumToStr(ERRNO, 0);
		Close logfile;
		TRYNEXT;
	ENDPROC

	!========================================
	! Test Runner
	!========================================
	PROC RunAllTests()
		TPWrite "Starting Robot2 Capabilities Test Suite...";
		TPWrite "";

		TestRobot2_ReadExternalAxes;
		WaitTime 2;

		TestRobot2_TCPCoordinates;
		WaitTime 2;

		TPWrite "";
		TPWrite "All tests complete!";
		TPWrite "Check /HOME folder for result files.";
	ENDPROC

	!========================================
	! Compare Robot1/Robot2 wobj0 (Snapshot)
	!========================================
	! Version: v1.6.0
	! Date: 2025-12-25
	! Purpose: Print Robot1/Robot2 wobj0 values and differences in one output
	PROC CompareWobj0Snapshots()
		VAR iodev logfile;
		VAR num dux;
		VAR num duy;
		VAR num duz;
		VAR num dox;
		VAR num doy;
		VAR num doz;
		VAR num duq1;
		VAR num duq2;
		VAR num duq3;
		VAR num duq4;
		VAR num doq1;
		VAR num doq2;
		VAR num doq3;
		VAR num doq4;

		TPWrite "========================================";
		TPWrite "Compare Robot1/Robot2 wobj0 (v1.6.0)";
		TPWrite "========================================";

		! Refresh Robot1 snapshot from TASK1
		%"T_ROB1:UpdateRobot1Wobj0Snapshot"%;

		TPWrite "Robot1 wobj0 (T_ROB1):";
		TPWrite "  UFrame X = " + NumToStr(robot1_wobj0_snapshot.uframe.trans.x, 2);
		TPWrite "  UFrame Y = " + NumToStr(robot1_wobj0_snapshot.uframe.trans.y, 2);
		TPWrite "  UFrame Z = " + NumToStr(robot1_wobj0_snapshot.uframe.trans.z, 2);
		TPWrite "  UFrame q1 = " + NumToStr(robot1_wobj0_snapshot.uframe.rot.q1, 4);
		TPWrite "  UFrame q2 = " + NumToStr(robot1_wobj0_snapshot.uframe.rot.q2, 4);
		TPWrite "  UFrame q3 = " + NumToStr(robot1_wobj0_snapshot.uframe.rot.q3, 4);
		TPWrite "  UFrame q4 = " + NumToStr(robot1_wobj0_snapshot.uframe.rot.q4, 4);
		TPWrite "  OFrame X = " + NumToStr(robot1_wobj0_snapshot.oframe.trans.x, 2);
		TPWrite "  OFrame Y = " + NumToStr(robot1_wobj0_snapshot.oframe.trans.y, 2);
		TPWrite "  OFrame Z = " + NumToStr(robot1_wobj0_snapshot.oframe.trans.z, 2);

		TPWrite "";
		TPWrite "Robot2 wobj0 (T_ROB2):";
		TPWrite "  UFrame X = " + NumToStr(wobj0.uframe.trans.x, 2);
		TPWrite "  UFrame Y = " + NumToStr(wobj0.uframe.trans.y, 2);
		TPWrite "  UFrame Z = " + NumToStr(wobj0.uframe.trans.z, 2);
		TPWrite "  UFrame q1 = " + NumToStr(wobj0.uframe.rot.q1, 4);
		TPWrite "  UFrame q2 = " + NumToStr(wobj0.uframe.rot.q2, 4);
		TPWrite "  UFrame q3 = " + NumToStr(wobj0.uframe.rot.q3, 4);
		TPWrite "  UFrame q4 = " + NumToStr(wobj0.uframe.rot.q4, 4);
		TPWrite "  OFrame X = " + NumToStr(wobj0.oframe.trans.x, 2);
		TPWrite "  OFrame Y = " + NumToStr(wobj0.oframe.trans.y, 2);
		TPWrite "  OFrame Z = " + NumToStr(wobj0.oframe.trans.z, 2);

		dux := wobj0.uframe.trans.x - robot1_wobj0_snapshot.uframe.trans.x;
		duy := wobj0.uframe.trans.y - robot1_wobj0_snapshot.uframe.trans.y;
		duz := wobj0.uframe.trans.z - robot1_wobj0_snapshot.uframe.trans.z;
		dox := wobj0.oframe.trans.x - robot1_wobj0_snapshot.oframe.trans.x;
		doy := wobj0.oframe.trans.y - robot1_wobj0_snapshot.oframe.trans.y;
		doz := wobj0.oframe.trans.z - robot1_wobj0_snapshot.oframe.trans.z;
		duq1 := wobj0.uframe.rot.q1 - robot1_wobj0_snapshot.uframe.rot.q1;
		duq2 := wobj0.uframe.rot.q2 - robot1_wobj0_snapshot.uframe.rot.q2;
		duq3 := wobj0.uframe.rot.q3 - robot1_wobj0_snapshot.uframe.rot.q3;
		duq4 := wobj0.uframe.rot.q4 - robot1_wobj0_snapshot.uframe.rot.q4;
		doq1 := wobj0.oframe.rot.q1 - robot1_wobj0_snapshot.oframe.rot.q1;
		doq2 := wobj0.oframe.rot.q2 - robot1_wobj0_snapshot.oframe.rot.q2;
		doq3 := wobj0.oframe.rot.q3 - robot1_wobj0_snapshot.oframe.rot.q3;
		doq4 := wobj0.oframe.rot.q4 - robot1_wobj0_snapshot.oframe.rot.q4;

		TPWrite "";
		TPWrite "Difference (R2 - R1):";
		TPWrite "  UFrame dX = " + NumToStr(dux, 2);
		TPWrite "  UFrame dY = " + NumToStr(duy, 2);
		TPWrite "  UFrame dZ = " + NumToStr(duz, 2);
		TPWrite "  UFrame dq1 = " + NumToStr(duq1, 4);
		TPWrite "  UFrame dq2 = " + NumToStr(duq2, 4);
		TPWrite "  UFrame dq3 = " + NumToStr(duq3, 4);
		TPWrite "  UFrame dq4 = " + NumToStr(duq4, 4);
		TPWrite "  OFrame dX = " + NumToStr(dox, 2);
		TPWrite "  OFrame dY = " + NumToStr(doy, 2);
		TPWrite "  OFrame dZ = " + NumToStr(doz, 2);
		TPWrite "  OFrame dq1 = " + NumToStr(doq1, 4);
		TPWrite "  OFrame dq2 = " + NumToStr(doq2, 4);
		TPWrite "  OFrame dq3 = " + NumToStr(doq3, 4);
		TPWrite "  OFrame dq4 = " + NumToStr(doq4, 4);
		TPWrite "========================================";

		Open "HOME:/wobj0_compare.txt", logfile \Write;
		Write logfile, "========================================";
		Write logfile, "Compare Robot1/Robot2 wobj0 (v1.6.0)";
		Write logfile, "========================================";
		Write logfile, "Date: " + CDate();
		Write logfile, "Time: " + CTime();
		Write logfile, "";
		Write logfile, "Robot1 wobj0 (T_ROB1):";
		Write logfile, "  UFrame X = " + NumToStr(robot1_wobj0_snapshot.uframe.trans.x, 2);
		Write logfile, "  UFrame Y = " + NumToStr(robot1_wobj0_snapshot.uframe.trans.y, 2);
		Write logfile, "  UFrame Z = " + NumToStr(robot1_wobj0_snapshot.uframe.trans.z, 2);
		Write logfile, "  UFrame q1 = " + NumToStr(robot1_wobj0_snapshot.uframe.rot.q1, 4);
		Write logfile, "  UFrame q2 = " + NumToStr(robot1_wobj0_snapshot.uframe.rot.q2, 4);
		Write logfile, "  UFrame q3 = " + NumToStr(robot1_wobj0_snapshot.uframe.rot.q3, 4);
		Write logfile, "  UFrame q4 = " + NumToStr(robot1_wobj0_snapshot.uframe.rot.q4, 4);
		Write logfile, "  OFrame X = " + NumToStr(robot1_wobj0_snapshot.oframe.trans.x, 2);
		Write logfile, "  OFrame Y = " + NumToStr(robot1_wobj0_snapshot.oframe.trans.y, 2);
		Write logfile, "  OFrame Z = " + NumToStr(robot1_wobj0_snapshot.oframe.trans.z, 2);
		Write logfile, "";
		Write logfile, "Robot2 wobj0 (T_ROB2):";
		Write logfile, "  UFrame X = " + NumToStr(wobj0.uframe.trans.x, 2);
		Write logfile, "  UFrame Y = " + NumToStr(wobj0.uframe.trans.y, 2);
		Write logfile, "  UFrame Z = " + NumToStr(wobj0.uframe.trans.z, 2);
		Write logfile, "  UFrame q1 = " + NumToStr(wobj0.uframe.rot.q1, 4);
		Write logfile, "  UFrame q2 = " + NumToStr(wobj0.uframe.rot.q2, 4);
		Write logfile, "  UFrame q3 = " + NumToStr(wobj0.uframe.rot.q3, 4);
		Write logfile, "  UFrame q4 = " + NumToStr(wobj0.uframe.rot.q4, 4);
		Write logfile, "  OFrame X = " + NumToStr(wobj0.oframe.trans.x, 2);
		Write logfile, "  OFrame Y = " + NumToStr(wobj0.oframe.trans.y, 2);
		Write logfile, "  OFrame Z = " + NumToStr(wobj0.oframe.trans.z, 2);
		Write logfile, "";
		Write logfile, "Difference (R2 - R1):";
		Write logfile, "  UFrame dX = " + NumToStr(dux, 2);
		Write logfile, "  UFrame dY = " + NumToStr(duy, 2);
		Write logfile, "  UFrame dZ = " + NumToStr(duz, 2);
		Write logfile, "  UFrame dq1 = " + NumToStr(duq1, 4);
		Write logfile, "  UFrame dq2 = " + NumToStr(duq2, 4);
		Write logfile, "  UFrame dq3 = " + NumToStr(duq3, 4);
		Write logfile, "  UFrame dq4 = " + NumToStr(duq4, 4);
		Write logfile, "  OFrame dX = " + NumToStr(dox, 2);
		Write logfile, "  OFrame dY = " + NumToStr(doy, 2);
		Write logfile, "  OFrame dZ = " + NumToStr(doz, 2);
		Write logfile, "  OFrame dq1 = " + NumToStr(doq1, 4);
		Write logfile, "  OFrame dq2 = " + NumToStr(doq2, 4);
		Write logfile, "  OFrame dq3 = " + NumToStr(doq3, 4);
		Write logfile, "  OFrame dq4 = " + NumToStr(doq4, 4);
		Write logfile, "========================================\0A";
		Close logfile;

		TPWrite "Saved to: /HOME/wobj0_compare.txt";

	ERROR
		TPWrite "ERROR in CompareWobj0Snapshots: " + NumToStr(ERRNO, 0);
		Close logfile;
		TRYNEXT;
	ENDPROC

	!========================================
	! Check wobj0 Definition
	!========================================
	! Version: v1.1.0
	! Date: 2025-12-18
	! Changes: Added file output to /HOME/task2_wobj0_definition.txt

	PROC ShowWobj0Definition()
		VAR string str_robhold;
		VAR string str_ufprog;
		VAR iodev logfile;

		TPWrite "========================================";
		TPWrite "TASK2 - wobj0 Definition (v1.1.0)";
		TPWrite "========================================";

		IF wobj0.robhold = TRUE THEN
			str_robhold := "TRUE";
		ELSE
			str_robhold := "FALSE";
		ENDIF

		IF wobj0.ufprog = TRUE THEN
			str_ufprog := "TRUE";
		ELSE
			str_ufprog := "FALSE";
		ENDIF

		TPWrite "wobj0.robhold: " + str_robhold;
		TPWrite "wobj0.ufprog: " + str_ufprog;
		TPWrite "";
		TPWrite "User Frame (uframe):";
		TPWrite "  X = " + NumToStr(wobj0.uframe.trans.x, 2) + " mm";
		TPWrite "  Y = " + NumToStr(wobj0.uframe.trans.y, 2) + " mm";
		TPWrite "  Z = " + NumToStr(wobj0.uframe.trans.z, 2) + " mm";
		TPWrite "  q1 = " + NumToStr(wobj0.uframe.rot.q1, 4);
		TPWrite "  q2 = " + NumToStr(wobj0.uframe.rot.q2, 4);
		TPWrite "  q3 = " + NumToStr(wobj0.uframe.rot.q3, 4);
		TPWrite "  q4 = " + NumToStr(wobj0.uframe.rot.q4, 4);
		TPWrite "";
		TPWrite "Object Frame (oframe):";
		TPWrite "  X = " + NumToStr(wobj0.oframe.trans.x, 2) + " mm";
		TPWrite "  Y = " + NumToStr(wobj0.oframe.trans.y, 2) + " mm";
		TPWrite "  Z = " + NumToStr(wobj0.oframe.trans.z, 2) + " mm";
		TPWrite "========================================";

		! Save to file
		Open "HOME:/task2_wobj0_definition.txt", logfile \Append;

		Write logfile, "========================================";
		Write logfile, "TASK2 - wobj0 Definition (v1.1.0)";
		Write logfile, "========================================";
		Write logfile, "Date: " + CDate();
		Write logfile, "Time: " + CTime();
		Write logfile, "";
		Write logfile, "wobj0.robhold: " + str_robhold;
		Write logfile, "wobj0.ufprog: " + str_ufprog;
		Write logfile, "";
		Write logfile, "User Frame (uframe):";
		Write logfile, "  X = " + NumToStr(wobj0.uframe.trans.x, 2) + " mm";
		Write logfile, "  Y = " + NumToStr(wobj0.uframe.trans.y, 2) + " mm";
		Write logfile, "  Z = " + NumToStr(wobj0.uframe.trans.z, 2) + " mm";
		Write logfile, "  q1 = " + NumToStr(wobj0.uframe.rot.q1, 4);
		Write logfile, "  q2 = " + NumToStr(wobj0.uframe.rot.q2, 4);
		Write logfile, "  q3 = " + NumToStr(wobj0.uframe.rot.q3, 4);
		Write logfile, "  q4 = " + NumToStr(wobj0.uframe.rot.q4, 4);
		Write logfile, "";
		Write logfile, "Object Frame (oframe):";
		Write logfile, "  X = " + NumToStr(wobj0.oframe.trans.x, 2) + " mm";
		Write logfile, "  Y = " + NumToStr(wobj0.oframe.trans.y, 2) + " mm";
		Write logfile, "  Z = " + NumToStr(wobj0.oframe.trans.z, 2) + " mm";
		Write logfile, "========================================\0A";

		Close logfile;
		TPWrite "Saved to: /HOME/task2_wobj0_definition.txt";

	ERROR
		TPWrite "ERROR in ShowWobj0Definition: " + NumToStr(ERRNO, 0);
		Close logfile;
		TRYNEXT;
	ENDPROC

	! Version: v1.1.0
	! Date: 2025-12-18
	! Changes: Added file output to /HOME/task2_world_vs_wobj0.txt

	PROC CompareWorldAndWobj0()
		VAR robtarget pos_world;
		VAR robtarget pos_wobj0;
		VAR iodev logfile;

		TPWrite "========================================";
		TPWrite "TASK2 - Compare World vs wobj0 (v1.1.0)";
		TPWrite "========================================";

		pos_world := CRobT(\Tool:=tool0);
		pos_wobj0 := CRobT(\Tool:=tool0\WObj:=wobj0);

		TPWrite "World Coordinates:";
		TPWrite "  X = " + NumToStr(pos_world.trans.x, 2) + " mm";
		TPWrite "  Y = " + NumToStr(pos_world.trans.y, 2) + " mm";
		TPWrite "  Z = " + NumToStr(pos_world.trans.z, 2) + " mm";
		TPWrite "";
		TPWrite "wobj0 Coordinates:";
		TPWrite "  X = " + NumToStr(pos_wobj0.trans.x, 2) + " mm";
		TPWrite "  Y = " + NumToStr(pos_wobj0.trans.y, 2) + " mm";
		TPWrite "  Z = " + NumToStr(pos_wobj0.trans.z, 2) + " mm";
		TPWrite "";
		TPWrite "Difference (World - wobj0):";
		TPWrite "  dX = " + NumToStr(pos_world.trans.x - pos_wobj0.trans.x, 2) + " mm";
		TPWrite "  dY = " + NumToStr(pos_world.trans.y - pos_wobj0.trans.y, 2) + " mm";
		TPWrite "  dZ = " + NumToStr(pos_world.trans.z - pos_wobj0.trans.z, 2) + " mm";
		TPWrite "========================================";

		! Save to file
		Open "HOME:/task2_world_vs_wobj0.txt", logfile \Append;

		Write logfile, "========================================";
		Write logfile, "TASK2 - Compare World vs wobj0 (v1.1.0)";
		Write logfile, "========================================";
		Write logfile, "Date: " + CDate();
		Write logfile, "Time: " + CTime();
		Write logfile, "";
		Write logfile, "World Coordinates:";
		Write logfile, "  X = " + NumToStr(pos_world.trans.x, 2) + " mm";
		Write logfile, "  Y = " + NumToStr(pos_world.trans.y, 2) + " mm";
		Write logfile, "  Z = " + NumToStr(pos_world.trans.z, 2) + " mm";
		Write logfile, "";
		Write logfile, "wobj0 Coordinates:";
		Write logfile, "  X = " + NumToStr(pos_wobj0.trans.x, 2) + " mm";
		Write logfile, "  Y = " + NumToStr(pos_wobj0.trans.y, 2) + " mm";
		Write logfile, "  Z = " + NumToStr(pos_wobj0.trans.z, 2) + " mm";
		Write logfile, "";
		Write logfile, "Difference (World - wobj0):";
		Write logfile, "  dX = " + NumToStr(pos_world.trans.x - pos_wobj0.trans.x, 2) + " mm";
		Write logfile, "  dY = " + NumToStr(pos_world.trans.y - pos_wobj0.trans.y, 2) + " mm";
		Write logfile, "  dZ = " + NumToStr(pos_world.trans.z - pos_wobj0.trans.z, 2) + " mm";
		Write logfile, "========================================\0A";

		Close logfile;
		TPWrite "Saved to: /HOME/task2_world_vs_wobj0.txt";

	ERROR
		TPWrite "ERROR in CompareWorldAndWobj0: " + NumToStr(ERRNO, 0);
		Close logfile;
		TRYNEXT;
	ENDPROC

	! ========================================
	! Verify TCP Orientation in All Coordinate Systems
	! ========================================
	! Version: v1.2.1
	! Date: 2025-12-19
	! Changes: Fixed "Too intense frequency of Write" error by adding WaitTime
	! Purpose: Compare TCP position and orientation in 4 coordinate systems:
	!   1. World - Global coordinate system
	!   2. wobj0 - Default work object (= World in current config)
	!   3. WobjFloor - Floor coordinate system at [-9500, 5300, 2100]
	!   4. wobjRob2Base - Robot2 Base Frame (45deg rotation per MOC.cfg)
	! Output: FlexPendant display + /HOME/task2_tcp_orientation.txt
	PROC VerifyTCPOrientation()
		VAR robtarget tcp_world;
		VAR robtarget tcp_wobj0;
		VAR robtarget tcp_floor;
		VAR robtarget tcp_rob_base;
		VAR iodev logfile;

		! Read TCP in all coordinate systems
		tcp_world := CRobT(\Tool:=tool0);
		tcp_wobj0 := CRobT(\Tool:=tool0\WObj:=wobj0);
		tcp_floor := CRobT(\Tool:=tool0\WObj:=WobjFloor);
		tcp_rob_base := CRobT(\Tool:=tool0\WObj:=wobjRob2Base);

		! Display on FlexPendant (reduced output)
		TPWrite "TASK2 - TCP Orientation (v1.2.1)";
		TPWrite "World: [" + NumToStr(tcp_world.trans.x, 1) + "," + NumToStr(tcp_world.trans.y, 1) + "," + NumToStr(tcp_world.trans.z, 1) + "]";
		TPWrite "Floor: [" + NumToStr(tcp_floor.trans.x, 1) + "," + NumToStr(tcp_floor.trans.y, 1) + "," + NumToStr(tcp_floor.trans.z, 1) + "]";
		TPWrite "Rob2Base: [" + NumToStr(tcp_rob_base.trans.x, 1) + "," + NumToStr(tcp_rob_base.trans.y, 1) + "," + NumToStr(tcp_rob_base.trans.z, 1) + "]";

		! Save to file (with WaitTime to prevent "Too intense frequency" error)
		Open "HOME:/task2_tcp_orientation.txt", logfile \Append;

		Write logfile, "========================================";
		Write logfile, "TASK2 - TCP Orientation Verification (v1.2.1)";
		Write logfile, "Date: " + CDate() + " " + CTime();
		Write logfile, "========================================";
		WaitTime 0.05;

		Write logfile, "1. World: Pos=[" + NumToStr(tcp_world.trans.x, 3) + "," + NumToStr(tcp_world.trans.y, 3) + "," + NumToStr(tcp_world.trans.z, 3) + "]";
		Write logfile, "   Rot=[" + NumToStr(tcp_world.rot.q1, 6) + "," + NumToStr(tcp_world.rot.q2, 6) + "," + NumToStr(tcp_world.rot.q3, 6) + "," + NumToStr(tcp_world.rot.q4, 6) + "]";
		WaitTime 0.05;

		Write logfile, "2. wobj0: Pos=[" + NumToStr(tcp_wobj0.trans.x, 3) + "," + NumToStr(tcp_wobj0.trans.y, 3) + "," + NumToStr(tcp_wobj0.trans.z, 3) + "]";
		Write logfile, "   Rot=[" + NumToStr(tcp_wobj0.rot.q1, 6) + "," + NumToStr(tcp_wobj0.rot.q2, 6) + "," + NumToStr(tcp_wobj0.rot.q3, 6) + "," + NumToStr(tcp_wobj0.rot.q4, 6) + "]";
		WaitTime 0.05;

		Write logfile, "3. Floor: Pos=[" + NumToStr(tcp_floor.trans.x, 3) + "," + NumToStr(tcp_floor.trans.y, 3) + "," + NumToStr(tcp_floor.trans.z, 3) + "]";
		Write logfile, "   Rot=[" + NumToStr(tcp_floor.rot.q1, 6) + "," + NumToStr(tcp_floor.rot.q2, 6) + "," + NumToStr(tcp_floor.rot.q3, 6) + "," + NumToStr(tcp_floor.rot.q4, 6) + "]";
		WaitTime 0.05;

		Write logfile, "4. Rob2Base: Pos=[" + NumToStr(tcp_rob_base.trans.x, 3) + "," + NumToStr(tcp_rob_base.trans.y, 3) + "," + NumToStr(tcp_rob_base.trans.z, 3) + "]";
		Write logfile, "   Rot=[" + NumToStr(tcp_rob_base.rot.q1, 6) + "," + NumToStr(tcp_rob_base.rot.q2, 6) + "," + NumToStr(tcp_rob_base.rot.q3, 6) + "," + NumToStr(tcp_rob_base.rot.q4, 6) + "]";
		WaitTime 0.05;

		Write logfile, "========================================\0A";

		Close logfile;
		TPWrite "Saved to: /HOME/task2_tcp_orientation.txt";

	ERROR
		TPWrite "ERROR in VerifyTCPOrientation: " + NumToStr(ERRNO, 0);
		Close logfile;
		TRYNEXT;
	ENDPROC

	! ========================================
	! Read TEST_MODE from /HOME/config.txt
	! ========================================
	! Returns: 0 if not found or error
	FUNC num ReadTestMode()
		VAR iodev configfile;
		VAR string line;
		VAR num test_mode;
		VAR bool found;
		VAR bool ok;
		VAR num line_count;
		VAR num max_lines;

		test_mode := 0;
		found := FALSE;
		line_count := 0;
		max_lines := 200;

		Open "HOME:/config.txt", configfile \Read;

		WHILE found = FALSE AND line_count < max_lines DO
			line := ReadStr(configfile \RemoveCR);
			line_count := line_count + 1;
			IF StrLen(line) = 0 THEN
				EXIT;
			ENDIF
			IF StrFind(line, 1, "TEST_MODE=") = 1 THEN
				IF StrLen(line) >= 11 THEN
					ok := StrToVal(StrPart(line, 11, StrLen(line) - 10), test_mode);
					found := TRUE;
				ENDIF
			ENDIF
		ENDWHILE

		Close configfile;
		RETURN test_mode;

	ERROR
		IF ERRNO = ERR_FILEOPEN THEN
			TPWrite "config.txt not found - using TEST_MODE=0";
		ENDIF
		Close configfile;
		RETURN 0;
	ENDFUNC

	! ========================================
	! Read Config Mode from /HOME/config.txt
	! ========================================
	! Version: v1.5.0
	! Date: 2025-12-24
	! Returns: 0 or 1 (default: 0 if file not found or error)
	FUNC num ReadConfigMode()
		VAR iodev configfile;
		VAR string line;
		VAR num mode_value;
		VAR bool found;
		VAR bool ok;

		mode_value := 0;  ! Default
		found := FALSE;

		! Try to open config.txt
		Open "HOME:/config.txt", configfile \Read;

		! Read lines until MODE= found
		WHILE found = FALSE DO
			line := ReadStr(configfile);

			! Check if line starts with "MODE="
			IF StrFind(line, 1, "MODE=") = 1 THEN
				! Extract number after "MODE=" (StrToVal returns bool, stores result in mode_value)
				ok := StrToVal(StrPart(line, 6, 1), mode_value);
				found := TRUE;
			ENDIF
		ENDWHILE

		Close configfile;
		RETURN mode_value;

	ERROR
		! File not found or read error - return default 0
		IF ERRNO = ERR_FILEOPEN THEN
			TPWrite "config.txt not found - using MODE=0";
		ENDIF
		Close configfile;
		RETURN 0;
	ENDFUNC

	! ========================================
	! Test Coordinate System Movement
	! ========================================
	! Version: v1.5.0
	! Date: 2025-12-24
	! Purpose: Verify coordinate system alignment by moving robot and comparing coordinates
	!   - Move robot in specified coordinate system
	!   - Check if Floor coordinate system shows expected movement
	!   - Validates coordinate system direction and position relationship
	! Parameters:
	!   delta_x, delta_y, delta_z: Movement distance (mm)
	!   mode: 0=WobjFloor base, 1=wobj0 base
	! Output: /HOME/task2_coordinate_test.txt
	PROC TestCoordinateMovement(num delta_x, num delta_y, num delta_z, num mode)
		VAR robtarget pos_start_wobj0;
		VAR robtarget pos_start_floor;
		VAR robtarget pos_target;
		VAR robtarget pos_end_wobj0;
		VAR robtarget pos_end_floor;
		VAR num diff_wobj0_x;
		VAR num diff_wobj0_y;
		VAR num diff_wobj0_z;
		VAR num diff_floor_x;
		VAR num diff_floor_y;
		VAR num diff_floor_z;
		VAR iodev logfile;

		! Read starting position in both coordinate systems
		pos_start_wobj0 := CRobT(\Tool:=tool0\WObj:=wobj0);
		pos_start_floor := CRobT(\Tool:=tool0\WObj:=WobjFloor);

		TPWrite "Start wobj0: [" + NumToStr(pos_start_wobj0.trans.x, 1) + "," + NumToStr(pos_start_wobj0.trans.y, 1) + "," + NumToStr(pos_start_wobj0.trans.z, 1) + "]";
		TPWrite "Start Floor: [" + NumToStr(pos_start_floor.trans.x, 1) + "," + NumToStr(pos_start_floor.trans.y, 1) + "," + NumToStr(pos_start_floor.trans.z, 1) + "]";

		! Calculate target position based on mode
		IF mode = 0 THEN
			! MODE=0: Use WobjFloor as base
			pos_target := CRobT(\Tool:=tool0\WObj:=WobjFloor);
			pos_target.trans.x := pos_target.trans.x + delta_x;
			pos_target.trans.y := pos_target.trans.y + delta_y;
			pos_target.trans.z := pos_target.trans.z + delta_z;
			TPWrite "Moving in Floor coordinate: [" + NumToStr(delta_x, 1) + "," + NumToStr(delta_y, 1) + "," + NumToStr(delta_z, 1) + "]";
			MoveL pos_target, v100, fine, tool0\WObj:=WobjFloor;
		ELSE
			! MODE=1: Use wobj0 as base
			pos_target := CRobT(\Tool:=tool0\WObj:=wobj0);
			pos_target.trans.x := pos_target.trans.x + delta_x;
			pos_target.trans.y := pos_target.trans.y + delta_y;
			pos_target.trans.z := pos_target.trans.z + delta_z;
			TPWrite "Moving in wobj0 coordinate: [" + NumToStr(delta_x, 1) + "," + NumToStr(delta_y, 1) + "," + NumToStr(delta_z, 1) + "]";
			MoveL pos_target, v100, fine, tool0\WObj:=wobj0;
		ENDIF

		! Read ending position in both coordinate systems
		pos_end_wobj0 := CRobT(\Tool:=tool0\WObj:=wobj0);
		pos_end_floor := CRobT(\Tool:=tool0\WObj:=WobjFloor);

		TPWrite "End wobj0: [" + NumToStr(pos_end_wobj0.trans.x, 1) + "," + NumToStr(pos_end_wobj0.trans.y, 1) + "," + NumToStr(pos_end_wobj0.trans.z, 1) + "]";
		TPWrite "End Floor: [" + NumToStr(pos_end_floor.trans.x, 1) + "," + NumToStr(pos_end_floor.trans.y, 1) + "," + NumToStr(pos_end_floor.trans.z, 1) + "]";

		! Calculate differences
		diff_wobj0_x := pos_end_wobj0.trans.x - pos_start_wobj0.trans.x;
		diff_wobj0_y := pos_end_wobj0.trans.y - pos_start_wobj0.trans.y;
		diff_wobj0_z := pos_end_wobj0.trans.z - pos_start_wobj0.trans.z;

		diff_floor_x := pos_end_floor.trans.x - pos_start_floor.trans.x;
		diff_floor_y := pos_end_floor.trans.y - pos_start_floor.trans.y;
		diff_floor_z := pos_end_floor.trans.z - pos_start_floor.trans.z;

		TPWrite "wobj0 moved: [" + NumToStr(diff_wobj0_x, 1) + "," + NumToStr(diff_wobj0_y, 1) + "," + NumToStr(diff_wobj0_z, 1) + "]";
		TPWrite "Floor moved: [" + NumToStr(diff_floor_x, 1) + "," + NumToStr(diff_floor_y, 1) + "," + NumToStr(diff_floor_z, 1) + "]";

		! Save to file
		Open "HOME:/task2_coordinate_test.txt", logfile \Append;

		Write logfile, "========================================";
		Write logfile, "TASK2 - Coordinate System Movement Test (v1.3.0)";
		Write logfile, "Date: " + CDate() + " " + CTime();
		Write logfile, "========================================";
		WaitTime 0.05;

		Write logfile, "Command: Move wobj0 [" + NumToStr(delta_x, 3) + "," + NumToStr(delta_y, 3) + "," + NumToStr(delta_z, 3) + "]";
		WaitTime 0.05;

		Write logfile, "Start wobj0: [" + NumToStr(pos_start_wobj0.trans.x, 3) + "," + NumToStr(pos_start_wobj0.trans.y, 3) + "," + NumToStr(pos_start_wobj0.trans.z, 3) + "]";
		Write logfile, "Start Floor: [" + NumToStr(pos_start_floor.trans.x, 3) + "," + NumToStr(pos_start_floor.trans.y, 3) + "," + NumToStr(pos_start_floor.trans.z, 3) + "]";
		WaitTime 0.05;

		Write logfile, "End wobj0: [" + NumToStr(pos_end_wobj0.trans.x, 3) + "," + NumToStr(pos_end_wobj0.trans.y, 3) + "," + NumToStr(pos_end_wobj0.trans.z, 3) + "]";
		Write logfile, "End Floor: [" + NumToStr(pos_end_floor.trans.x, 3) + "," + NumToStr(pos_end_floor.trans.y, 3) + "," + NumToStr(pos_end_floor.trans.z, 3) + "]";
		WaitTime 0.05;

		Write logfile, "wobj0 moved: [" + NumToStr(diff_wobj0_x, 3) + "," + NumToStr(diff_wobj0_y, 3) + "," + NumToStr(diff_wobj0_z, 3) + "]";
		Write logfile, "Floor moved: [" + NumToStr(diff_floor_x, 3) + "," + NumToStr(diff_floor_y, 3) + "," + NumToStr(diff_floor_z, 3) + "]";
		WaitTime 0.05;

		Write logfile, "Verification: If wobj0 and Floor have same direction,";
		Write logfile, "  movement should be identical in both coordinate systems.";
		Write logfile, "========================================\0A";

		Close logfile;
		TPWrite "Saved to: /HOME/task2_coordinate_test.txt";

	ERROR
		TPWrite "ERROR in TestCoordinateMovement: " + NumToStr(ERRNO, 0);
		Close logfile;
		TRYNEXT;
	ENDPROC

	! ========================================
	! Move to Safe Middle Position
	! ========================================
	! Version: v1.4.0
	! Date: 2025-12-23
	! Purpose: Move gantry to middle of stroke range for safe testing
	! Middle positions: M1=1.4m, M2=2.65m, M3=0.5m
	PROC MoveToMiddlePosition()
		VAR jointtarget middle_pos;

		TPWrite "Moving to middle position...";

		middle_pos := CJointT();

		! Set gantry axes to middle positions (safe testing position)
		middle_pos.extax.eax_a := 1400;     ! M1DM3 middle: (-9.51+12.31)/2 = 1.4m = 1400mm
		middle_pos.extax.eax_b := 2650;     ! M2DM3 middle: (-0.05+5.35)/2 = 2.65m = 2650mm
		middle_pos.extax.eax_c := 500;      ! M3DM3 middle: (-0.05+1.05)/2 = 0.5m = 500mm

		MoveAbsJ middle_pos, v100, fine, tool0;

		TPWrite "Reached middle position";
	ENDPROC

	! ========================================
	! Test Gantry Axis Movement
	! ========================================
	! Version: v1.4.0
	! Date: 2025-12-23
	! Purpose: Move gantry joint axes and compare wobj0 vs Floor coordinate changes
	! Parameters:
	!   delta_m1 - M1DM3 (X axis) movement in mm
	!   delta_m2 - M2DM3 (Y axis) movement in mm
	!   delta_m3 - M3DM3 (Z axis) movement in mm
	PROC TestGantryAxisMovement(num delta_m1, num delta_m2, num delta_m3)
		VAR jointtarget joints_start;
		VAR jointtarget joints_end;
		VAR robtarget tcp_start_wobj0;
		VAR robtarget tcp_end_wobj0;
		VAR robtarget tcp_start_floor;
		VAR robtarget tcp_end_floor;
		VAR num wobj0_dx;
		VAR num wobj0_dy;
		VAR num wobj0_dz;
		VAR num floor_dx;
		VAR num floor_dy;
		VAR num floor_dz;
		VAR iodev logfile;

		! Read starting positions
		joints_start := CJointT();
		tcp_start_wobj0 := CRobT(\Tool:=tool0\WObj:=wobj0);
		tcp_start_floor := CRobT(\Tool:=tool0\WObj:=WobjFloor);

		TPWrite "Start - Gantry: M1=" + NumToStr(joints_start.extax.eax_a, 1) + " M2=" + NumToStr(joints_start.extax.eax_b, 1) + " M3=" + NumToStr(joints_start.extax.eax_c, 1);

		! Calculate target joint position
		joints_end := joints_start;
		joints_end.extax.eax_a := joints_end.extax.eax_a + delta_m1;
		joints_end.extax.eax_b := joints_end.extax.eax_b + delta_m2;
		joints_end.extax.eax_c := joints_end.extax.eax_c + delta_m3;

